# B&R Automation Studio project 8238 (part 11)

```iecst
			//###DK2012Jan12
			// Set statistic.
			IF _wPrevMsgStatisticSelect <> IFmnMsg.In.wMsgStatisticSelect THEN
				_wPrevMsgStatisticSelect := IFmnMsg.In.wMsgStatisticSelect;
				_xMsgStatisticSelectChanged := TRUE;
			END_IF;

			IF IFmnMsg.Trig.xRefreshStatistic OR _xRefreshStatistic THEN
				_msgStatisticNumShowIdx := _msgStatisticNumIdx;
				_msgStatisticTimeShowIdx := _msgStatisticTimeIdx;
				_wIFMsgStatisticCntNumShow := _wIFMsgStatisticCntNum;
				_wIFMsgStatisticCntTimeShow := _wIFMsgStatisticCntTime;
				IFmnMsg.Trig.xRefreshStatistic := FALSE;
				_xRefreshStatistic := FALSE;
				_xMsgStatisticSelectChanged := TRUE;
			END_IF;

			IF _xMsgStatisticSelectChanged THEN
				IF IFmnMsg.In.wMsgStatisticSelect = 0 THEN
					IFmnMsg.Out.wMsgStatisticCnt := _wIFMsgStatisticCntNumShow;
					FOR _wMsgListCnt := 0 TO MNMSG_MAX_IDX_VCMSGSTATLIST BY 1 DO
						_utfMsgTextTempFirst := UINT_TO_WSTRING(_msgStatisticNumShowIdx[_wMsgListCnt].wFunction_ID);
						_utfMsgTextTempSecond := ".";
						brwcsncat(ADR(_utfMsgTextTempFirst), ADR(_utfMsgTextTempSecond),
						UDINT_TO_UINT(brwcslen(ADR(_utfMsgTextTempSecond)) - (brwcslen(ADR(_utfMsgTextTempFirst)) + brwcslen(ADR(_utfMsgTextTempSecond)) - (SIZEOF(_utfMsgTextTempFirst) / 2 - 1))));
						_utfMsgTextTempSecond := UINT_TO_WSTRING(_msgStatisticNumShowIdx[_wMsgListCnt].wMsgNumber);
						brwcsncat(ADR(_utfMsgTextTempFirst), ADR(_utfMsgTextTempSecond),
						UDINT_TO_UINT(brwcslen(ADR(_utfMsgTextTempSecond)) - (brwcslen(ADR(_utfMsgTextTempFirst)) + brwcslen(ADR(_utfMsgTextTempSecond)) - (SIZEOF(_utfMsgTextTempFirst) / 2 - 1))));
						_utfMsgTextTempSecond := ".";
						brwcsncat(ADR(_utfMsgTextTempFirst), ADR(_utfMsgTextTempSecond),
						UDINT_TO_UINT(brwcslen(ADR(_utfMsgTextTempSecond)) - (brwcslen(ADR(_utfMsgTextTempFirst)) + brwcslen(ADR(_utfMsgTextTempSecond)) - (SIZEOF(_utfMsgTextTempFirst) / 2 - 1))));
						_utfMsgTextTempSecond := UINT_TO_WSTRING(_msgStatisticNumShowIdx[_wMsgListCnt].wInstance);
						brwcsncat(ADR(_utfMsgTextTempFirst), ADR(_utfMsgTextTempSecond),
						UDINT_TO_UINT(brwcslen(ADR(_utfMsgTextTempSecond)) - (brwcslen(ADR(_utfMsgTextTempFirst)) + brwcslen(ADR(_utfMsgTextTempSecond)) - (SIZEOF(_utfMsgTextTempFirst) / 2 - 1))));
						_utfMsgTextTempSecond := " ";
						brwcsncat(ADR(_utfMsgTextTempFirst), ADR(_utfMsgTextTempSecond),
						UDINT_TO_UINT(brwcslen(ADR(_utfMsgTextTempSecond)) - (brwcslen(ADR(_utfMsgTextTempFirst)) + brwcslen(ADR(_utfMsgTextTempSecond)) - (SIZEOF(_utfMsgTextTempFirst) / 2 - 1))));
						_wActFunctionID := _msgStatisticNumShowIdx[_wMsgListCnt].wFunction_ID;
						_wActMsgNumber := _msgStatisticNumShowIdx[_wMsgListCnt].wMsgNumber;
						_wActInstance := _msgStatisticNumShowIdx[_wMsgListCnt].wInstance;
						_actGetTxtFim;
						IF NOT((_wActFunctionID = 0) OR (_wActMsgNumber = 0)) THEN
							IFmnMsg.Out.MsgStatistic[_wMsgListCnt].utfMsgText := _utfMsgTextTempFirst;
							IFmnMsg.Out.MsgStatistic[_wMsgListCnt].lValue := _msgStatisticNumShowIdx[_wMsgListCnt].lValue;
						ELSE
							IFmnMsg.Out.MsgStatistic[_wMsgListCnt].utfMsgText := "";
							IFmnMsg.Out.MsgStatistic[_wMsgListCnt].lValue := 0;
						END_IF;
					END_FOR;
				END_IF;
				IF IFmnMsg.In.wMsgStatisticSelect = 1 THEN
					IFmnMsg.Out.wMsgStatisticCnt := _wIFMsgStatisticCntTimeShow;
					FOR _wMsgListCnt := 0 TO MNMSG_MAX_IDX_VCMSGSTATLIST BY 1 DO
						_utfMsgTextTempFirst := UINT_TO_WSTRING(_msgStatisticTimeShowIdx[_wMsgListCnt].wFunction_ID);
						_utfMsgTextTempSecond := ".";
						brwcsncat(ADR(_utfMsgTextTempFirst), ADR(_utfMsgTextTempSecond),
						UDINT_TO_UINT(brwcslen(ADR(_utfMsgTextTempSecond)) - (brwcslen(ADR(_utfMsgTextTempFirst)) + brwcslen(ADR(_utfMsgTextTempSecond)) - (SIZEOF(_utfMsgTextTempFirst) / 2 - 1))));
						_utfMsgTextTempSecond := UINT_TO_WSTRING(_msgStatisticTimeShowIdx[_wMsgListCnt].wMsgNumber);
						brwcsncat(ADR(_utfMsgTextTempFirst), ADR(_utfMsgTextTempSecond),
						UDINT_TO_UINT(brwcslen(ADR(_utfMsgTextTempSecond)) - (brwcslen(ADR(_utfMsgTextTempFirst)) + brwcslen(ADR(_utfMsgTextTempSecond)) - (SIZEOF(_utfMsgTextTempFirst) / 2 - 1))));
						_utfMsgTextTempSecond := ".";
						brwcsncat(ADR(_utfMsgTextTempFirst), ADR(_utfMsgTextTempSecond),
						UDINT_TO_UINT(brwcslen(ADR(_utfMsgTextTempSecond)) - (brwcslen(ADR(_utfMsgTextTempFirst)) + brwcslen(ADR(_utfMsgTextTempSecond)) - (SIZEOF(_utfMsgTextTempFirst) / 2 - 1))));
						_utfMsgTextTempSecond := UINT_TO_WSTRING(_msgStatisticTimeShowIdx[_wMsgListCnt].wInstance);
						brwcsncat(ADR(_utfMsgTextTempFirst), ADR(_utfMsgTextTempSecond),
						UDINT_TO_UINT(brwcslen(ADR(_utfMsgTextTempSecond)) - (brwcslen(ADR(_utfMsgTextTempFirst)) + brwcslen(ADR(_utfMsgTextTempSecond)) - (SIZEOF(_utfMsgTextTempFirst) / 2 - 1))));
						_utfMsgTextTempSecond := " ";
						brwcsncat(ADR(_utfMsgTextTempFirst), ADR(_utfMsgTextTempSecond),
						UDINT_TO_UINT(brwcslen(ADR(_utfMsgTextTempSecond)) - (brwcslen(ADR(_utfMsgTextTempFirst)) + brwcslen(ADR(_utfMsgTextTempSecond)) - (SIZEOF(_utfMsgTextTempFirst) / 2 - 1))));
						_wActFunctionID := _msgStatisticTimeShowIdx[_wMsgListCnt].wFunction_ID;
						_wActMsgNumber := _msgStatisticTimeShowIdx[_wMsgListCnt].wMsgNumber;
						_wActInstance := _msgStatisticTimeShowIdx[_wMsgListCnt].wInstance;
						_actGetTxtFim;
						IF NOT ((_wActFunctionID = 0) OR (_wActMsgNumber = 0)) THEN
							IFmnMsg.Out.MsgStatistic[_wMsgListCnt].utfMsgText := _utfMsgTextTempFirst;
							IFmnMsg.Out.MsgStatistic[_wMsgListCnt].lValue := _msgStatisticTimeShowIdx[_wMsgListCnt].lValue;
						ELSE
							IFmnMsg.Out.MsgStatistic[_wMsgListCnt].utfMsgText := "";
							IFmnMsg.Out.MsgStatistic[_wMsgListCnt].lValue := 0;
						END_IF;
					END_FOR;
				END_IF;
				_xMsgStatisticSelectChanged := FALSE;
			END_IF;
			//###DK2012Jan12

		END_IF

	ELSE	// _Plausibility.xOK

		// Horning for 500ms. After it has finished it will start again ten seconds later.
		_tonCrit1(IN := NOT _tonCrit2.Q, PT := T#500ms);
		_tonCrit2(IN := _tonCrit1.Q, PT := T#10s);

		IFmnMsg.Out.bHorn := SEL(NOT _tonCrit1.Q, 0, 1);	// Causes some horning now.

		IFmnMsg.Out.bLight := 1;

		// Meldung setzen

		IF _xNotOkFirstScan THEN

			_xNotOkFirstScan := FALSE;

			// Meldungsliste füllen

			brsmemset (ADR(mnMsgStatAd.Msg), 0, SIZEOF (mnMsgStatAd.Msg));

			_InsertMsgLine.AdrIntFaultList := ADR(mnMsgStatAd.Msg.MsgListFaultInt);
			_InsertMsgLine.AdrCntIntFault := ADR(mnMsgStatAd.Msg.MsgCntFaultInt);

			_dtHelp(enable := TRUE);

			_InsertMsgLine.Class := MNMSG_CLASS_INTFAULT;
			_InsertMsgLine.Insert := TRUE;
			_InsertMsgLine.MsgLine.bAckLevel := MNMSG_CLASS_NO_ACK;
			_InsertMsgLine.MsgLine.bInstance := 0;
			_InsertMsgLine.MsgLine.diAttr1 := 0;
			_InsertMsgLine.MsgLine.wFunction_ID := 2;
			_InsertMsgLine.MsgLine.wMsgNumber := MNMSG_MSG_SYSTEMFAULT;
			_InsertMsgLine.MsgLine.TimeStamp := _dtHelp.DT1;
			_InsertMsgLine();

			mnMsgStatAd.Msg.dtMsgIntFaultChanged := _dtHelp.DT1;

		END_IF

	END_IF;	// IFmnMsg.Out.xMnMsgReady

	////////////////////////////////////////////////////////////////////////////////////////////////////////////////////////////////////////////////////////////////////////////////////////////////////////////////////////////////////////////////////////////////////////////////////////////////////////////////////////////////////////////////////////////////////////////////////////////////////////////////////////////////////////////////////////////////////////////////////////////////////////////////////////////////////////////////////////////////////////////////////////////////////////////////////////////////////

	_LastExecute(enable := TRUE);
	_dtLastExecute := _LastExecute.DT1;

END_PROGRAM
```

#### mnMsgInit.st - Initialization code
```iecst
(********************************************************************
 * COPYRIGHT -- Herbert Kannegiesser GmbH
 ********************************************************************
 * Program: mnMsg
 * File: mnMsgInit.st
 * Author: subramaniam/hunholz
 * Created: January 28, 2011
 * Changed: October 20, 2011 by A. Hunholz
 ********************************************************************
 * Implementation of program mnMsg
 ********************************************************************
*)
PROGRAM _INIT

	// Packet-Version auslesen mit MO_ver aus SYS_lib und für den Additional Status zur Verfügung stellen

	_sPkgName := 'mnMsg';

	IF ( MO_ver(ADR(_sPkgName), 0, ADR(_VerStruc)) = 0 ) THEN

		brsmemcpy(ADR(mnMsgStatAd.sPkgVersion), ADR(_VerStruc.version), SIZEOF(_VerStruc.version));

	ELSE

		mnMsgStatAd.sPkgVersion := '---';

	END_IF

	//********************Startoption der Plausibilitaetspruefung**********************
	//____________________________________________________________

	// Initialisierung von (Zaehl)variablen und Booleans
	_xMsgStatisticNumFirstEntry 	:= TRUE;
	_xMsgStatisticWriteNum 			:= TRUE;
	_xMsgStatisticTimeFirstEntry 	:= TRUE;
	_xMsgStatisticWriteTime 		:= TRUE;
	_xFirstElementToInsertTime 		:= TRUE;
	_xFirstElementToInsertNum 		:= TRUE;

	// Filter setzen
	IFmnMsg.In.wMsgHistListClassSelect.0 := 1;
	IFmnMsg.In.wMsgHistListClassSelect.1 := 1;
	IFmnMsg.In.wMsgHistListClassSelect.2 := 1;
	IFmnMsg.In.wMsgHistListClassSelect.3 := 1;

	_EventStatisticDelStep := Del_Wait;

	//*********************Synchrone Schnittstelle zurücksetzen*****************************

	brsmemset(ADR(IFmnMsg.Out),0,SIZEOF(IFmnMsg.Out));
	brsmemset (ADR (kgMsgStatus[MNMSG_IDX_KGMSGSTAT]), 0, SIZEOF (kgMsgStatus[0]));

	//*********************Alle Listen loeschen

	brsmemset (ADR(_MsgImage), 0, SIZEOF (_MsgImage));	// Meldungsabbild
	brsmemset (ADR(_MsgImageState),0,SIZEOF(_MsgImageState));	// Meldungsabbild

	brsmemset (ADR(mnMsgStatAd.Msg), 0 ,SIZEOF (mnMsgStatAd.Msg));

	//****************************************************************************************************************
	// Log erzeugen
	//****************************************************************************************************************

	_kgArLogWrite.enable := TRUE;
	_kgArLogWrite.ident := 0;
	_kgArLogWrite.errornr := 50001;

	_AsArLogCreate(enable := TRUE, pName := ADR('mnMsgL'), len := 4096, memType := arlogUSRROM);

	IF _AsArLogCreate.status = ERR_OK THEN

		_kgArLogWrite.ident := _AsArLogCreate.ident;

	ELSIF _AsArLogCreate.status = arlogERR_EXISTING THEN

		_AsArLogGetInfo(enable := TRUE, pName := ADR('mnMsgL'));

		IF _AsArLogGetInfo.status = ERR_OK THEN

			_kgArLogWrite.ident := _AsArLogGetInfo.ident;

		END_IF

	END_IF

	//***************** Datenobjekte prüfen
	//______________________________

	// Unbedingtes REPEAT, damit bei Fehler alles Andere per EXIT
	// übersprungen werden kann.

	REPEAT

		//*************** KONFIGURATION
		//**************************************
		// _doInfoCfg 'Bild der Konfigurationsdatei' of DatObjInfo

		_doInfoCfg.enable := TRUE;	// VAR_INPUT BOOL enable 'enables execution'
		_doInfoCfg.pName := ADR('CfgMsgStat');	// VAR_INPUT UDINT pName 'name of data object'
		_doInfoCfg();

		IF _doInfoCfg.status <> ERR_OK THEN

			_kgArLogWrite.logLevel := arlogLEVEL_INFO;
			_kgArLogWrite.text := 'Messageconfiguration does not exist: {##AttrVar1}';
			_kgArLogWrite.var1 := _doInfoCfg.status;
			_kgArLogWrite.var2 := 0;
			_kgArLogWrite();
			EXIT;

		ELSE

			// _doInfoCfg 'Bild der Konfigurationsdatei' of DatObjInfo
			// wCntCfg of Plausib_Typ: number of configuration entries
			_Plausibility.dCfgLen := _doInfoCfg.len; // VAR_OUTPUT UDINT len 'length of the data area in the data object'
			_Plausibility.dCfgMem := _doInfoCfg.pDatObjMem; // VAR_OUTPUT UDINT pDatObjMem 'pointer to the data in the data object'
			_Plausibility.wCfgCnt := UDINT_TO_UINT((_doInfoCfg.len-SIZEOF(UINT))/SIZEOF (MsgCfgLine_Typ)); // Laenge der Version zu Beginn abziehen

			_wVersion ACCESS _Plausibility.dCfgMem;
			_Plausibility.wCfgVersion := _wVersion;

			IF _Plausibility.wCfgCnt > MNMSG_MAX_CFGMESSAGES THEN

				_kgArLogWrite.logLevel := arlogLEVEL_INFO;
				_kgArLogWrite.text := 'To much entries in Messageconfiguration: {##AttrVar1}';
				_kgArLogWrite.var1 := _Plausibility.wCfgCnt;
				_kgArLogWrite.var2 := 0;
				_kgArLogWrite();
				EXIT;

			END_IF

			// Zugriff auf die Konfigurationszeilen
			_MsgCfgList ACCESS _doInfoCfg.pDatObjMem + SIZEOF(UINT); // Offset Versionsnummer

			// Binäre Suche initialisieren
			_BinSearchCfg.MsgCfgList := _doInfoCfg.pDatObjMem + SIZEOF(UINT);	// Offset Versionsnummer
			_BinSearchCfg.wCntMsgCfg := _Plausibility.wCfgCnt;	// VAR_INPUT UINT wCntMsgCfg

		END_IF

		//*****************************
		// STATISTIK
		//*****************************

		_kgCheckStat(Enable := TRUE, pName := ADR('_MsgStat'), MinLen := SIZEOF(_MsgStatList), NomLen := SIZEOF(_MsgStatList), Create := TRUE, MemType := doUSRROM);

		IF _kgCheckStat.Status = ERR_OK OR _kgCheckStat.Status = KG_INFO_DO_NEW THEN

			_doWriteStat.enable := TRUE;
			_doWriteStat.ident := _kgCheckStat.doId;

			IF _kgCheckStat.Status = KG_INFO_DO_NEW THEN

				// Kopfdaten schreiben
				_StatHeader.lVersion := _Plausibility.wCfgVersion;
				_StatHeader.lLength :=  UINT_TO_UDINT(MNMSG_MAX_CFGMESSAGES);

				_doWriteStat.Offset := 0;
				_doWriteStat.len := SIZEOF(_StatHeader);
				_doWriteStat.pSource := ADR(_StatHeader);
				_doWriteStat();

				IF _doWriteStat.status = ERR_OK THEN

					_xStatReady := TRUE;
					_MsgStatList ACCESS _kgCheckStat.doMem;

					_kgArLogWrite.logLevel := arlogLEVEL_INFO;
					_kgArLogWrite.text := 'Statistic created!';
					_kgArLogWrite.var1 := 0;
					_kgArLogWrite.var2 := 0;
					_kgArLogWrite();

				ELSE

					_kgArLogWrite.logLevel := arlogLEVEL_INFO;
					_kgArLogWrite.text := 'Write Statistic: {##AttrVar1}';
					_kgArLogWrite.var1 := _doWriteStat.status;
					_kgArLogWrite.var2 := 0;
					_kgArLogWrite();

				END_IF

			ELSE

				brsmemcpy(ADR(_StatHeader), _kgCheckStat.doMem, SIZEOF(_StatHeader));

				IF _StatHeader.lVersion <> _Plausibility.wCfgVersion THEN

					//Konfigurationsversion hat sich geändert --> Statistik neu erstellen

					_doDeleteStat(enable := TRUE, ident := _kgCheckStat.doId);

					_kgCheckStat(Enable := TRUE, pName := ADR('_MsgStat'), MinLen := SIZEOF(_MsgStatList), NomLen := SIZEOF(_MsgStatList), Create := TRUE, MemType := doUSRROM);

					IF _kgCheckStat.Status = KG_INFO_DO_NEW THEN

						_doWriteStat.enable := TRUE;
						_doWriteStat.ident := _kgCheckStat.doId;

						// Kopfdaten schreiben
						_StatHeader.lVersion := _Plausibility.wCfgVersion;
						_StatHeader.lLength :=  UINT_TO_UDINT(MNMSG_MAX_CFGMESSAGES);

						_doWriteStat.Offset := 0;
						_doWriteStat.len := SIZEOF(_StatHeader);
						_doWriteStat.pSource := ADR(_StatHeader);
						_doWriteStat();

						IF _doWriteStat.status = ERR_OK THEN

							_xStatReady := TRUE;
							_MsgStatList ACCESS _kgCheckStat.doMem;

							_kgArLogWrite.logLevel := arlogLEVEL_INFO;
							_kgArLogWrite.text := 'Statistic recreated!';
							_kgArLogWrite.var1 := 0;
							_kgArLogWrite.var2 := 0;
							_kgArLogWrite();

						ELSE

							_kgArLogWrite.logLevel := arlogLEVEL_INFO;
							_kgArLogWrite.text := 'Write Statistic*: {##AttrVar1}';
							_kgArLogWrite.var1 := _doWriteStat.status;
							_kgArLogWrite.var2 := 0;
							_kgArLogWrite();

						END_IF

					ELSE

						_kgArLogWrite.logLevel := arlogLEVEL_INFO;
						_kgArLogWrite.text := 'Check Statistic*: {##AttrVar1}';
						_kgArLogWrite.var1 := _kgCheckStat.Status;
						_kgArLogWrite.var2 := 0;
						_kgArLogWrite();

					END_IF

				ELSE //IF _StatHeader.lVersion <> _Plausibility.wCfgVersion THEN

					// Version ist OK
					_xStatReady := TRUE;
					_MsgStatList ACCESS _kgCheckStat.doMem;

				END_IF

			END_IF

		ELSE

			_kgArLogWrite.logLevel := arlogLEVEL_INFO;
			_kgArLogWrite.text := 'Check Statistic: {##AttrVar1}';
			_kgArLogWrite.var1 := _kgCheckStat.Status;
			_kgArLogWrite.var2 := 0;
			_kgArLogWrite();

		END_IF

		//*************** RINGBUFFER
		//*********************************

		_kgCheckHist(Enable := TRUE, pName := ADR('_MsgRB'), MinLen :=  MNMSG_MAX_MESSAGEHISTORY * SIZEOF(MsgHistList_Typ), NomLen :=  MNMSG_MAX_MESSAGEHISTORY * SIZEOF(MsgHistList_Typ), Create := TRUE, MemType := doUSRROM);

		IF _kgCheckHist.Status = ERR_OK OR _kgCheckHist.Status = KG_INFO_DO_NEW THEN

			IF _kgCheckHist.Status = KG_INFO_DO_NEW THEN

				_kgArLogWrite.logLevel := arlogLEVEL_INFO;
				_kgArLogWrite.text := 'History created!';
				_kgArLogWrite.var1 := 0;
				_kgArLogWrite.var2 := 0;
				_kgArLogWrite();

				_wPtrRBwrite := 0;
				_wPtrRBread := 0;
				_wPtrRBloc := 0;

			END_IF

			_xRBReady := TRUE;

			// _InsertRB of msgInsertRB 'Eintrag in den Ringbuffer'
			_InsertRB.doIdent := _kgCheckHist.doId;
			_InsertRB.doLen := _kgCheckHist.doLen;

			_ReadRB.doIdent := _kgCheckHist.doId;
			_ReadRB.doLen := _kgCheckHist.doLen;

			_LocRB.doIdent := _kgCheckHist.doId;
			_LocRB.doLen := _kgCheckHist.doLen;

			_DebugHistory ACCESS _kgCheckHist.doMem;

		ELSE

			_kgArLogWrite.logLevel := arlogLEVEL_INFO;
			_kgArLogWrite.text := 'Check History: {##AttrVar1}';
			_kgArLogWrite.var1 := _kgCheckStat.Status;
			_kgArLogWrite.var2 := 0;
			_kgArLogWrite();

		END_IF

		_Plausibility.xOK := TRUE;

		//***********************************************************************************
		// Statistik für Werte vor dem letzten Ausschalten schreiben, um dann die
		// Statistik zurücksetzen zu können
		//***********************************************************************************

		IF _xRBReady THEN

			FOR _wMsgIdx := 1 TO _Plausibility.wCfgCnt DO

				IF _MsgImageTime[_wMsgIdx].dtTimeStamp <> DT#1970-01-01-00:00:00  THEN

					// Es steht noch eine Zeit im Image, die noch nicht erfasst wurde
					// D.h. beim Ausschalten der SPS stand diese Meldung noch an.

					_lTime := 0;

					IF _xStatReady THEN

						// Statistik schreiben
						IF (_dtLastExecute >= _MsgImageTime[_wMsgIdx].dtTimeStamp) THEN
							_lTime := DiffDT(_dtLastExecute, _MsgImageTime[_wMsgIdx].dtTimeStamp);
						END_IF

						_StatLine.lTime := _MsgStatList.List[_wMsgIdx].lTime + _lTime;
						_StatLine.lCnt := _MsgStatList.List[_wMsgIdx].lCnt + 1;
						_StatLine.wFunction_ID := _MsgCfgList[_wMsgIdx].wFunction_ID;
						_StatLine.wMsgNumber := _MsgCfgList[_wMsgIdx].wMsgNumber;
						_StatLine.wInstance := _MsgCfgList[_wMsgIdx].wInstance;
						_StatLine.wMsgClass := _MsgStatList.List[_wMsgIdx].wMsgClass;

						_doWriteStat.Offset := SIZEOF(_StatHeader) + (_wMsgIdx-1)*SIZEOF(_StatLine);
						_doWriteStat.len := SIZEOF(_StatLine);
						_doWriteStat.pSource := ADR(_StatLine);

						_doWriteStat();

					END_IF

					// Ringbuffer schreiben
					_TempHistline.TimeStampEvent := _dtLastExecute;
					_TempHistline.wFunction_ID := _MsgCfgList[_wMsgIdx].wFunction_ID;
					_TempHistline.wInstance := _MsgCfgList[_wMsgIdx].wInstance;
					_TempHistline.wMsgNumber := _MsgCfgList[_wMsgIdx].wMsgNumber;
					IF _xStatReady THEN
						_TempHistline.wMsgClass := _MsgStatList.List[_wMsgIdx].wMsgClass;
					ELSE
						_TempHistline.wMsgClass := MNMSG_CLASS_INFO;
					END_IF
					_TempHistline.diAttr1 := 0;
					_TempHistline.diAttr2 := 0;
					_TempHistline.sAttrTxt := '';
					_TempHistline.wEvent := MNMSG_EVENT_GONE;	// Constant of library KGlibMMsg UINT MSG_EVENT_GONE = 3
					_TempHistline.lTime := _lTime;

					_InsertRB.pEntry := ADR(_TempHistline);
					_InsertRB.lLenEntry := SIZEOF(_TempHistline);
					_InsertRB(wPtrWrite := _wPtrRBwrite, wPtrRead := _wPtrRBread, wPtrStart := _wPtrRBstart);

					IF _InsertRB.wStatus <> ERR_OK THEN
						_kgArLogWrite.logLevel := arlogLEVEL_INFO;
						_kgArLogWrite.text := 'Inster History: {##AttrVar1}';
						_kgArLogWrite.var1 := _InsertRB.wStatus;
						_kgArLogWrite.var2 := 0;
						_kgArLogWrite();
					END_IF

				END_IF

			END_FOR

		END_IF

		// Nachdem das Image in die Statistik und in den Ringbuffer geschrieben wurde,
		// kann es auf Null zurückgesetzt werden
		brsmemset(ADR(_MsgImageTime),0,SIZEOF(_MsgImageTime));

		UNTIL

		TRUE

	END_REPEAT;

	_dtHelp(enable := TRUE);

	_xStatFault := NOT _xStatReady;

	_xNotOkFirstScan := TRUE;

END_PROGRAM
```

#### mnMsg.typ - Local data types
```iecst
(********************************************************************
 * COPYRIGHT -- Herbert Kannegiesser GmbH
 ********************************************************************
 * Program: mnMsg
 * File: mnMsg.typ
 * Author: subramaniam/Hunholz
 * Created: January 28, 2011
 * Changed: June 15, 2011
 ********************************************************************
 * Local data types of program mnMsg
 ********************************************************************)

TYPE
	CmdState_enum :
		(
		enCS_Idle,
		enCS_WaitForZero,
		enCS_CmdDelStat,
		enCS_CmdDelHist
		);
	EventStatisticDel_enum :
		(
		Del_Delete,
		Del_Wait,
		Del_Check,
		Del_Write,
		Del_Error
		);
	EventHistDel_enum :
		(
		Del_DeleteH,
		Del_WaitH,
		Del_ErrorH
		);
END_TYPE

(*Plausibilitaetspruefung Meldungsmanager ----------------------------------------------------------------------------------------------------------------------------------------------------------------------------------------*)

TYPE
	Plausib_Typ : 	STRUCT
		dCfgMem : UDINT;
		dCfgLen : UDINT;
		wCfgCnt : UINT;
		wCfgVersion : UINT;
		xOK : BOOL;
	END_STRUCT;
END_TYPE

(*Meldungsabbild ----------------------------------------------------------------------------------------------------------------------------------------------------------------------------------------*)

TYPE
	ImageMsgState_Typ : 	STRUCT
		xOn : BOOL;
		xChanged : BOOL;
	END_STRUCT;
	ImageMsgTime_Typ : 	STRUCT
		dtTimeStamp : DATE_AND_TIME;
	END_STRUCT;
	ImageMsg_Typ : 	STRUCT
		wStatus : UINT;
		wMsgClass : UINT;
		wMsgAckLevel : UINT;
		sMsgAttrTxt : STRING[13];
		diMsgAttr1 : DINT;
		diMsgAttr2 : DINT;
	END_STRUCT;
	ImageMsgHelp_Typ : 	STRUCT  (*Hilfsstruktur der Meldeabbild*)
		xFaultIntChanged : BOOL;
		xFaultExtChanged : BOOL;
		xWarningChanged : BOOL;
		xInfoChanged : BOOL;
		xMaintChanged : BOOL;
	END_STRUCT;
	mnMsgStatisticIdx_Type : 	STRUCT
		wFunction_ID : UINT;
		wMsgNumber : UINT;
		wInstance : UINT;
		lValue : UDINT;
	END_STRUCT;
END_TYPE
```

#### mnMsg.var - Local variables
```iecst
(********************************************************************
 * COPYRIGHT -- Herbert Kannegiesser GmbH
 ********************************************************************
 * Program: mnMsg
 * File: mnMsg.var
 * Author: subramaniam/hunholz
 * Created: January 28, 2011
 * Changed: June 15, 2011
 ********************************************************************
 * Local variables of program mnMsg
 ********************************************************************)
(*Plausibilitaetspruefung Meldungsmanager *)
VAR
	_Plausibility : Plausib_Typ := (dCfgMem:=0,dCfgLen:=0,wCfgCnt:=0,wCfgVersion:=0,xOK:=FALSE);
	_xTrigRefreshHistList : BOOL;
	_lErrCnt : UDINT;
	_TONrepeatDFII : TON;
END_VAR
(*Meldungsabbild *)
VAR
	_MsgImage : ARRAY[1..MNMSG_MAX_CFGMESSAGES] OF ImageMsg_Typ;
	_MsgImageState : ARRAY[1..MNMSG_MAX_CFGMESSAGES] OF ImageMsgState_Typ;
	_MsgImageHelp : ImageMsgHelp_Typ;
END_VAR
VAR RETAIN
	_MsgImageTime : ARRAY[1..MNMSG_MAX_CFGMESSAGES] OF ImageMsgTime_Typ;
END_VAR
(* Bild der Konfigurationsdatei *)
VAR
	_doInfoCfg : DatObjInfo;
	_MsgCfgList : REFERENCE TO ARRAY[1..MNMSG_MAX_CFGMESSAGES] OF MsgCfgLine_Typ;
END_VAR
(*Bild der Textdatei*)
(* In diesem Fall, wird die Länge des Arrays nicht von mnTxt bestimmt *)
VAR
	_MsgTxtLine : REFERENCE TO ARRAY[1..MNMSG_MAX_CFGMESSAGES] OF MsgTxtLine_Typ;
	_MsgHelpTxtLine : REFERENCE TO ARRAY[1..MNMSG_MAX_CFGMESSAGES] OF MsgHelpTxtLine_Typ;
END_VAR
(* Bild der Statistikdatei*)
VAR
	_MsgStatList : REFERENCE TO MsgStat_Typ;
END_VAR
(*Bild der Text-Meldungshistorie*)
VAR
	_MsgHistListRB : ARRAY[0..MNMSG_MAX_IDX_VCMSGHISTLIST] OF IFmnMsgOutMsgHistList_Typ;
END_VAR
(*Interne Meldung*)
VAR
	_mnMsgStat : kgMsg_Status_Typ := (0);
END_VAR
(*Kommandbefehle *)
(*  Zeiger auf Zusatzattribute *)
VAR
	_iCmdData0 : REFERENCE TO ARRAY[0..1] OF UINT;
	_iCmdData1 : REFERENCE TO ARRAY[0..1] OF UINT;
END_VAR
(*Schnittstelle Visualisierung für Ringbuffer und Statistik *)
VAR
	_xAck : BOOL;
	_wCntFaultNotAck : UINT;
	_xCmdAckAll : BOOL;
	_xCmdAck : BOOL;
	_xCmdAckAllMaint : BOOL;
END_VAR
(*Letzte Ausführungszeit bestimmen*)
VAR
	_LastExecute : DTGetTime;
END_VAR
VAR RETAIN
	_dtLastExecute : DATE_AND_TIME := 0;
END_VAR
(*Aktueller Zeitstempel*)
VAR
	_dtTimeStamp : DTGetTime;
END_VAR
(* Binäre Suche *)
VAR
	_BinSearchCfg : msgBinSearchCfgList;
	_BinSearchTxt : msgBinSearchTxtLine;
	_BinSearchHelpTxt : msgBinSearchHelpTxtLine;
END_VAR
(*Suche*)
VAR
	_GetNextChrPos : msgNextChrPos;
END_VAR
(* Ringbuffer *)
VAR
	_InsertRB : kgRBinsert;
	_ReadRB : kgRBread;
	_LocRB : kgRBloc;
	_wStepRdRb : UINT;
	_xRBReady : BOOL := FALSE;
	_xMnTxtReady : BOOL := FALSE;
END_VAR
VAR RETAIN
	_wPtrRBwrite : UINT;
	_wPtrRBread : UINT;
	_wPtrRBloc : UINT;
	_wPtrRBstart : UINT;
END_VAR
(* Statistik*)
VAR
	_StatLine : MsgStatList_Typ;
	_StatHeader : MsgStatHeader_Typ;
	_doWriteStat : DatObjWrite;
	_doDeleteStat : DatObjDelete;
	_xStatReady : BOOL := FALSE;
END_VAR
(* Meldungslisten *)
VAR
	_InsertMsgLine : msgInsertMsgLine;
END_VAR
(* Hupensteuerung *)
VAR
	_xHornFaultOn : BOOL;
	_xHornWarnOn : BOOL;
	_tpFault : TP;
	_tonFault1 : TON;
	_tonFault2 : TON;
	_xHornFaultOnh : BOOL;
	_xHornWarnOnh : BOOL;
	_tpWarn : TP;
	_tonWarn2 : TON;
	_tonWarn1 : TON;
	_wFaultMode : UINT;
	_wWarnMode : UINT;
END_VAR
(*MsgStatistic*)
VAR
	_msgStatisticNumIdx : ARRAY[0..MNMSG_MAX_IDX_VCMSGSTATLIST] OF mnMsgStatisticIdx_Type;
	_msgStatisticTimeIdx : ARRAY[0..MNMSG_MAX_IDX_VCMSGSTATLIST] OF mnMsgStatisticIdx_Type;
	_msgStatisticNumShowIdx : ARRAY[0..MNMSG_MAX_IDX_VCMSGSTATLIST] OF mnMsgStatisticIdx_Type;
	_msgStatisticTimeShowIdx : ARRAY[0..MNMSG_MAX_IDX_VCMSGSTATLIST] OF mnMsgStatisticIdx_Type;
END_VAR
(* Hilfsvariablen *)
VAR
	_wSrcIdx : UDINT;
	_wMsgIdx : UINT;
	_wTxtIdx : UINT;
	_wImageIdx : UINT;
	_lTime : UDINT;
	_ii : UINT;
	_dtHelp : DTGetTime;
	_xMnParOk : BOOL := FALSE;
	_xMsgClassChanged : BOOL := FALSE;
	_xAckLevelChanged : BOOL;
	_xAckLevelRosen : BOOL := FALSE;
	_xAckLevelFallen : BOOL := FALSE;
	_EventStatisticDelStep : EventStatisticDel_enum;
	_EventHistDelStep : EventHistDel_enum;
	_tonCrit1 : TON;
	_tonCrit2 : TON;
END_VAR
VAR CONSTANT
	MSW : UINT := 1; (*Most Significant Word*)
	LSW : UINT := 0; (*Leas Significant Word*)
END_VAR
VAR
	_enIFCmdState : CmdState_enum := enCS_Idle;
	_enExtCmdState : CmdState_enum := enCS_Idle;
	_xIFcmdHornOff : BOOL := FALSE;
	_wMsgListCnt : UINT;
	_wIFMsgListCnt : UINT;
	_wIFMsgStatisticCntTime : UINT;
	_wIFMsgStatisticCntNum : UINT;
	_wIFMsgStatisticCntTimeShow : UINT;
	_wIFMsgStatisticCntNumShow : UINT;
	_xMsgStatisticNumFirstEntry : BOOL;
	_xMsgStatisticWriteNum : BOOL;
	_xMsgStatisticTimeFirstEntry : BOOL;
	_xMsgStatisticWriteTime : BOOL;
	_wPosMinTime : UINT;
	_wPosMinNum : UINT;
	_wPosMaxTime : UINT;
	_wPosMaxNum : UINT;
	_wPosEndTime : UINT;
	_wPosEndNum : UINT;
	_wPosSearchTime : UINT;
	_wPosSearchNum : UINT;
	_diMemMoveTimeIdx : DINT := 0;
	_diMemMoveNumIdx : DINT := 0;
	_xPosFoundTime : BOOL;
	_xPosFoundNum : BOOL;
	_xFirstElementToInsertTime : BOOL;
	_xFirstElementToInsertNum : BOOL;
	_lValueNumMin : UDINT;
	_lValueTimeMin : UDINT;
	_lValueTime : UDINT;
	_lValueNum : UDINT;
	_wPrevMsgStatisticSelect : UINT := 0;
	_xMsgStatisticSelectChanged : BOOL := FALSE;
	_utfMsgTextTempFirst : WSTRING[67];
	_utfMsgTextTempSecond : WSTRING[255];
	_utfMsgTextTempThird : WSTRING[255];
	_utfMsgTextTempFourth : WSTRING[255];
	_fbMsgReplSubStr : msgReplSubStr;
	_lHElseTime1 : UDINT := 0;
	_lHElseTime2 : UDINT := 0;
	_lHElseTime3 : UDINT := 0;
	_lHElseTime3EndPos : UDINT := 0;
	_wHElseTime3PosSearch : UINT := 0;
	_lHElseTime3lValuePosP0 : UDINT := 0;
	_lHElseTime3lValuePosP1 : UDINT := 0;
	_lHElseTime3lValueTime : UDINT := 0;
	_lHElseNum1 : UDINT := 0;
	_lHElseNum2 : UDINT := 0;
	_lHElseNum3 : UDINT := 0;
	_TempHistline : MsgHistList_Typ;
	_kgArLogWrite : kgArLogWrite;
	_AsArLogCreate : AsArLogCreate;
	_AsArLogGetInfo : AsArLogGetInfo;
	_xLogNoCfg : BOOL;
	_xLogCfgMoved : BOOL;
END_VAR
VAR CONSTANT
	MNMSG_MSG_NO_MESSAGE : UINT := 0;
END_VAR
VAR
	_xStatFault : BOOL;
	_xLogDeleteStat : BOOL;
	_xLogCreateStat : BOOL;
	_xLogInfoStat : BOOL;
	_xLogWriteStat : BOOL;
	_wPrevLCID : UINT := 0;
	_xUpdateMsgList : BOOL := FALSE;
	_xUpdateMsgHistListRB : BOOL := FALSE;
	_wMsgHistListCntUpdate : UINT := 0;
	_utfMsgTxtLCIDfirst : WSTRING[67];
	_utfMsgTxtLCIDsecond : WSTRING[67];
	_utfRbsDateTime : WSTRING[67];
	_utfLCIDFunctionId : WSTRING[67];
	_utfLCIDMsgNumber : WSTRING[67];
	_utfLCIDInstance : WSTRING[67];
	_wLCIDFunctionId : UINT;
	_wLCIDMsgNumber : UINT;
	_wLCIDInstance : UINT;
	_lPosPointFirst : UDINT;
	_lPosPointSecond : UDINT;
	_lPosSpaceFirst : UDINT;
	_lPosSpaceSecond : UDINT;
	_lAdrPointFirst : UDINT;
	_lAdrPointSecond : UDINT;
	_lAdrSpaceFirst : UDINT;
	_lAdrSpaceSecond : UDINT;
	_wCntSafety : UINT := 0;
	_sPkgName : STRING[10];
	_VerStruc : MoVerStruc_typ;
	_wPrevMsgHistListOffsetRB : UINT;
	_wMsgHistListOffsetRB : UINT;
	_xRefreshHistListRB : BOOL;
	_xMsgHistListOffsetChRB : BOOL;
	_wPrevMsgHistListEventSelRB : UINT;
	_wMsgHistListEventSelRB : UINT;
	_xMsgHistListEventSelChRB : BOOL;
	_wPrevMsgHistListClassSelRB : UINT;
	_wMsgHistListClassSelRB : UINT;
	_xMsgHistListClassSelChRB : BOOL;
	_xMsgHistListPointToMinRB : BOOL;
	_wPtrRBlocTemp : UINT;
	_wPtrRBlocTempTwo : UINT;
	_wPtrRBlocTempThree : UINT;
	_wPtrRBlocTempFour : UINT;
	_xPtrRBlocAgain : BOOL;
	_wPtrRBlocLastFound : UINT;
	_wMsgHistListMaxOffsetRB : UINT;
	_xTrigPrevMsgHistListPageRB : BOOL;
	_xTrigNextMsgHistListPageRB : BOOL;
	_xRBoneTurn : BOOL;
	_wMsgHistListCntRB : UINT;
	_wActFunctionID : UINT;
	_wActMsgNumber : UINT;
	_diActAttr1 : DINT;
	_diActAttr2 : DINT;
	_sActAttrTxt : STRING[13];
	_wActInstance : UINT;
	_wActEvent : UINT;
	_lActTime : UDINT;
	_bActMsgLClass : USINT;
	_xSelOk : BOOL;
	_xTurnaround : BOOL;
	_xExtCmdAckAll : BOOL;
	_xExtCmdAck : BOOL;
	_xExtCmdAckAllMaint : BOOL;
	_wExtCmdFunctionID : UINT;
	_wExtCmdMsgNo : UINT;
	_wExtCmdInstance : UINT;
	_wExtCmdAckLevel : UINT;
	_xExtcmdHornOff : BOOL;
	_xDeleteMsgStat : BOOL;
	_wMsgCntMaint : UINT;
	_wIdxMsgListMaint : UINT;
	_xUpdateMsgListLan : BOOL;
	_xRefreshStatistic : BOOL;
	_xRefreshHistList : BOOL;
	_wLCID : UINT;
	_kgCheckStat : kgCheckDo;
	_kgCheckHist : kgCheckDo;
	_wVersion : REFERENCE TO UINT;
	_wLogStep : UINT;
	_xNotOkFirstScan : BOOL;
	_DebugHistory : REFERENCE TO ARRAY[0..MNMSG_MAX_MESSAGEHISTORY] OF MsgHistList_Typ;
END_VAR
```

#### _actGetTxtFim.st
```iecst
(********************************************************************
 * COPYRIGHT -- Herbert Kannegiesser GmbH
 ********************************************************************
 * Program: mnMsg
 * File: actGetTxtFim.st
 * Author: kuehne
 * Created: February 21, 2012
 ********************************************************************
 * Implementation of program mnMsg
 ********************************************************************)

(* Add a new action to your IEC program or library *)
ACTION _actGetTxtFim:
	IF _xMnTxtReady THEN
		_MsgTxtLine ACCESS IFmnTxt.Out.ptrFunctionTxtList;
		_BinSearchTxt.MsgTxtList := IFmnTxt.Out.ptrFunctionTxtList;
		_BinSearchTxt.wCntMsgTxt := IFmnTxt.Out.wCntFunctionTxt;
		_BinSearchTxt.wFunctionID := _wActFunctionID;
		_BinSearchTxt.wNumber := _wActMsgNumber;
		_BinSearchTxt.wInstance := _wActInstance;
		_BinSearchTxt.bTupel := 1;
		_BinSearchTxt();
		IF _BinSearchTxt.wStatus <> ERR_OK THEN
			brwcscat(ADR(_utfMsgTextTempFirst), ADR(""));
		ELSE
			_wTxtIdx := _BinSearchTxt.wMsgPos;
			_BinSearchCfg.wFunctionID := _wActFunctionID;
			_BinSearchCfg.wMsgNo := _wActMsgNumber;
			_BinSearchCfg.wInstance := _wActInstance;
			_BinSearchCfg();
			IF _BinSearchCfg.wStatus = ERR_OK THEN
				_wImageIdx := _BinSearchCfg.wMsgIdx;
				_utfMsgTextTempThird := "";
				_utfMsgTextTempThird := DINT_TO_WSTRING(_MsgImage[_wImageIdx].diMsgAttr1);
			ELSE
				_utfMsgTextTempThird := "{##AttrVar1}";
			END_IF;
			_utfMsgTextTempSecond := "";
			_fbMsgReplSubStr.utfStr := ADR(_MsgTxtLine[_wTxtIdx].utfText);
			_fbMsgReplSubStr.utfSubStr := ADR("{##AttrVar1}");
			_fbMsgReplSubStr.utfStrToReplWith := ADR(_utfMsgTextTempThird);
			_fbMsgReplSubStr.utfStrResult := ADR(_utfMsgTextTempSecond);
			_fbMsgReplSubStr();
			IF _BinSearchCfg.wStatus = ERR_OK THEN
				_wImageIdx := _BinSearchCfg.wMsgIdx;
				_utfMsgTextTempThird := "";
				_utfMsgTextTempThird := DINT_TO_WSTRING(_MsgImage[_wImageIdx].diMsgAttr2);
			ELSE
				_utfMsgTextTempThird := "{##AttrVar2}";
			END_IF;
			_utfMsgTextTempFourth := "";
			_utfMsgTextTempFourth := _utfMsgTextTempSecond;
			_utfMsgTextTempSecond := "";
			_fbMsgReplSubStr.utfStr := ADR(_utfMsgTextTempFourth);
			_fbMsgReplSubStr.utfSubStr := ADR("{##AttrVar2}");
			_fbMsgReplSubStr.utfStrToReplWith := ADR(_utfMsgTextTempThird);
			_fbMsgReplSubStr.utfStrResult := ADR(_utfMsgTextTempSecond);
			_fbMsgReplSubStr();
			IF _BinSearchCfg.wStatus = ERR_OK THEN
				_wImageIdx := _BinSearchCfg.wMsgIdx;
				_utfMsgTextTempThird := "";
				_utfMsgTextTempThird := STRING_TO_WSTRING(_MsgImage[_wImageIdx].sMsgAttrTxt);
			ELSE
				_utfMsgTextTempThird := "{##AttrTxt}";
			END_IF;
			_utfMsgTextTempFourth := "";
			_utfMsgTextTempFourth := _utfMsgTextTempSecond;
			_utfMsgTextTempSecond := "";
			_fbMsgReplSubStr.utfStr := ADR(_utfMsgTextTempFourth);
			_fbMsgReplSubStr.utfSubStr := ADR("{##AttrTxt}");
			_fbMsgReplSubStr.utfStrToReplWith := ADR(_utfMsgTextTempThird);
			_fbMsgReplSubStr.utfStrResult := ADR(_utfMsgTextTempSecond);
			_fbMsgReplSubStr();
			brwcsncat(ADR(_utfMsgTextTempFirst), ADR(_utfMsgTextTempSecond),
			UDINT_TO_UINT(brwcslen(ADR(_utfMsgTextTempSecond)) - (brwcslen(ADR(_utfMsgTextTempFirst)) + brwcslen(ADR(_utfMsgTextTempSecond)) - (SIZEOF(_utfMsgTextTempFirst) / 2 - 1))));
			_utfMsgTextTempSecond := "";
			_utfMsgTextTempSecond := ": ";
			brwcsncat(ADR(_utfMsgTextTempFirst), ADR(_utfMsgTextTempSecond),
			UDINT_TO_UINT(brwcslen(ADR(_utfMsgTextTempSecond)) - (brwcslen(ADR(_utfMsgTextTempFirst)) + brwcslen(ADR(_utfMsgTextTempSecond)) - (SIZEOF(_utfMsgTextTempFirst) / 2 - 1))));
		END_IF;
		_MsgTxtLine ACCESS IFmnTxt.Out.ptrInstanceTxtList;
		_BinSearchTxt.MsgTxtList := IFmnTxt.Out.ptrInstanceTxtList;
		_BinSearchTxt.wCntMsgTxt := IFmnTxt.Out.wCntInstanceTxt;
		_BinSearchTxt.wFunctionID := _wActFunctionID;
		_BinSearchTxt.wNumber := _wActInstance;
		_BinSearchTxt.wInstance := 0;
		_BinSearchTxt.bTupel := 2;
		_BinSearchTxt();
		IF _BinSearchTxt.wStatus <> ERR_OK THEN
			brwcscat(ADR(_utfMsgTextTempFirst), ADR(""));
		ELSE
			_wTxtIdx := _BinSearchTxt.wMsgPos;
			_BinSearchCfg.wFunctionID := _wActFunctionID;
			_BinSearchCfg.wMsgNo := _wActMsgNumber;
			_BinSearchCfg.wInstance := _wActInstance;
			_BinSearchCfg();
			IF _BinSearchCfg.wStatus = ERR_OK THEN
				_wImageIdx := _BinSearchCfg.wMsgIdx;
				_utfMsgTextTempThird := "";
				_utfMsgTextTempThird := DINT_TO_WSTRING(_MsgImage[_wImageIdx].diMsgAttr1);
			ELSE
				_utfMsgTextTempThird := "{##AttrVar1}";
			END_IF;
			_utfMsgTextTempSecond := "";
			_fbMsgReplSubStr.utfStr := ADR(_MsgTxtLine[_wTxtIdx].utfText);
			_fbMsgReplSubStr.utfSubStr := ADR("{##AttrVar1}");
			_fbMsgReplSubStr.utfStrToReplWith := ADR(_utfMsgTextTempThird);
			_fbMsgReplSubStr.utfStrResult := ADR(_utfMsgTextTempSecond);
			_fbMsgReplSubStr();
			IF _BinSearchCfg.wStatus = ERR_OK THEN
				_wImageIdx := _BinSearchCfg.wMsgIdx;
				_utfMsgTextTempThird := "";
				_utfMsgTextTempThird := DINT_TO_WSTRING(_MsgImage[_wImageIdx].diMsgAttr2);
			ELSE
				_utfMsgTextTempThird := "{##AttrVar2}";
			END_IF;
			_utfMsgTextTempFourth := "";
			_utfMsgTextTempFourth := _utfMsgTextTempSecond;
			_utfMsgTextTempSecond := "";
			_fbMsgReplSubStr.utfStr := ADR(_utfMsgTextTempFourth);
			_fbMsgReplSubStr.utfSubStr := ADR("{##AttrVar2}");
			_fbMsgReplSubStr.utfStrToReplWith := ADR(_utfMsgTextTempThird);
			_fbMsgReplSubStr.utfStrResult := ADR(_utfMsgTextTempSecond);
			_fbMsgReplSubStr();
			IF _BinSearchCfg.wStatus = ERR_OK THEN
				_wImageIdx := _BinSearchCfg.wMsgIdx;
				_utfMsgTextTempThird := "";
				_utfMsgTextTempThird := STRING_TO_WSTRING(_MsgImage[_wImageIdx].sMsgAttrTxt);
			ELSE
				_utfMsgTextTempThird := "{##AttrTxt}";
			END_IF;
			_utfMsgTextTempFourth := "";
			_utfMsgTextTempFourth := _utfMsgTextTempSecond;
			_utfMsgTextTempSecond := "";
			_fbMsgReplSubStr.utfStr := ADR(_utfMsgTextTempFourth);
			_fbMsgReplSubStr.utfSubStr := ADR("{##AttrTxt}");
			_fbMsgReplSubStr.utfStrToReplWith := ADR(_utfMsgTextTempThird);
			_fbMsgReplSubStr.utfStrResult := ADR(_utfMsgTextTempSecond);
			_fbMsgReplSubStr();
			brwcsncat(ADR(_utfMsgTextTempFirst), ADR(_utfMsgTextTempSecond),
			UDINT_TO_UINT(brwcslen(ADR(_utfMsgTextTempSecond)) - (brwcslen(ADR(_utfMsgTextTempFirst)) + brwcslen(ADR(_utfMsgTextTempSecond)) - (SIZEOF(_utfMsgTextTempFirst) / 2 - 1))));
			_utfMsgTextTempSecond := "";
			_utfMsgTextTempSecond := ": ";
			brwcsncat(ADR(_utfMsgTextTempFirst), ADR(_utfMsgTextTempSecond),
			UDINT_TO_UINT(brwcslen(ADR(_utfMsgTextTempSecond)) - (brwcslen(ADR(_utfMsgTextTempFirst)) + brwcslen(ADR(_utfMsgTextTempSecond)) - (SIZEOF(_utfMsgTextTempFirst) / 2 - 1))));
		END_IF;
		_MsgTxtLine ACCESS IFmnTxt.Out.ptrMessageTxtList;
		_BinSearchTxt.MsgTxtList := IFmnTxt.Out.ptrMessageTxtList;
		_BinSearchTxt.wCntMsgTxt := IFmnTxt.Out.wCntMessageTxt;
		_BinSearchTxt.wFunctionID := _wActFunctionID;
		_BinSearchTxt.wNumber := _wActMsgNumber;
		_BinSearchTxt.wInstance := _wActInstance;
		_BinSearchTxt.bTupel := 2;
		_BinSearchTxt();
		IF _BinSearchTxt.wStatus <> ERR_OK THEN
			brwcscat(ADR(_utfMsgTextTempFirst), ADR(""));
		ELSE
			_wTxtIdx := _BinSearchTxt.wMsgPos;
			_BinSearchCfg.wFunctionID := _wActFunctionID;
			_BinSearchCfg.wMsgNo := _wActMsgNumber;
			_BinSearchCfg.wInstance := _wActInstance;
			_BinSearchCfg();
			IF _BinSearchCfg.wStatus = ERR_OK THEN
				_wImageIdx := _BinSearchCfg.wMsgIdx;
				_utfMsgTextTempThird := "";
				_utfMsgTextTempThird := DINT_TO_WSTRING(_MsgImage[_wImageIdx].diMsgAttr1);
			ELSE
				_utfMsgTextTempThird := "{##AttrVar1}";
			END_IF;
			_utfMsgTextTempSecond := "";
			_fbMsgReplSubStr.utfStr := ADR(_MsgTxtLine[_wTxtIdx].utfText);
			_fbMsgReplSubStr.utfSubStr := ADR("{##AttrVar1}");
			_fbMsgReplSubStr.utfStrToReplWith := ADR(_utfMsgTextTempThird);
			_fbMsgReplSubStr.utfStrResult := ADR(_utfMsgTextTempSecond);
			_fbMsgReplSubStr();
			IF _BinSearchCfg.wStatus = ERR_OK THEN
				_wImageIdx := _BinSearchCfg.wMsgIdx;
				_utfMsgTextTempThird := "";
				_utfMsgTextTempThird := DINT_TO_WSTRING(_MsgImage[_wImageIdx].diMsgAttr2);
			ELSE
				_utfMsgTextTempThird := "{##AttrVar2}";
			END_IF;
			_utfMsgTextTempFourth := "";
			_utfMsgTextTempFourth := _utfMsgTextTempSecond;
			_utfMsgTextTempSecond := "";
			_fbMsgReplSubStr.utfStr := ADR(_utfMsgTextTempFourth);
			_fbMsgReplSubStr.utfSubStr := ADR("{##AttrVar2}");
			_fbMsgReplSubStr.utfStrToReplWith := ADR(_utfMsgTextTempThird);
			_fbMsgReplSubStr.utfStrResult := ADR(_utfMsgTextTempSecond);
			_fbMsgReplSubStr();
			IF _BinSearchCfg.wStatus = ERR_OK THEN
				_wImageIdx := _BinSearchCfg.wMsgIdx;
				_utfMsgTextTempThird := "";
				_utfMsgTextTempThird := STRING_TO_WSTRING(_MsgImage[_wImageIdx].sMsgAttrTxt);
			ELSE
				_utfMsgTextTempThird := "{##AttrTxt}";
			END_IF;
			_utfMsgTextTempFourth := "";
			_utfMsgTextTempFourth := _utfMsgTextTempSecond;
			_utfMsgTextTempSecond := "";
			_fbMsgReplSubStr.utfStr := ADR(_utfMsgTextTempFourth);
			_fbMsgReplSubStr.utfSubStr := ADR("{##AttrTxt}");
			_fbMsgReplSubStr.utfStrToReplWith := ADR(_utfMsgTextTempThird);
			_fbMsgReplSubStr.utfStrResult := ADR(_utfMsgTextTempSecond);
			_fbMsgReplSubStr();
			brwcsncat(ADR(_utfMsgTextTempFirst), ADR(_utfMsgTextTempSecond),
			UDINT_TO_UINT(brwcslen(ADR(_utfMsgTextTempSecond)) - (brwcslen(ADR(_utfMsgTextTempFirst)) + brwcslen(ADR(_utfMsgTextTempSecond)) - (SIZEOF(_utfMsgTextTempFirst) / 2 - 1))));
		END_IF;
	ELSE
		brwcscat(ADR(_utfMsgTextTempFirst), ADR(""));
	END_IF;
END_ACTION
```

#### _actGetTxtFimh.st
```iecst
(********************************************************************
 * COPYRIGHT -- Herbert Kannegiesser GmbH
 ********************************************************************
 * Program: mnMsg
 * File: actGetTxtFimh.st
 * Author: kuehne
 * Created: February 22, 2012
 ********************************************************************
 * Implementation of program mnMsg
 ********************************************************************)

 (* Add a new action to your IEC program or library *)
ACTION _actGetTxtFimh:
	IF _xMnTxtReady THEN
		_MsgTxtLine ACCESS IFmnTxt.Out.ptrFunctionTxtList;
		_BinSearchTxt.MsgTxtList := IFmnTxt.Out.ptrFunctionTxtList;
		_BinSearchTxt.wCntMsgTxt := IFmnTxt.Out.wCntFunctionTxt;
		_BinSearchTxt.wFunctionID := _wActFunctionID;
		_BinSearchTxt.wNumber := _wActMsgNumber;
		_BinSearchTxt.wInstance := _wActInstance;
		_BinSearchTxt.bTupel := 1;
		_BinSearchTxt();
		IF _BinSearchTxt.wStatus <> ERR_OK THEN
			brwcscat(ADR(_utfMsgTextTempFirst), ADR(""));
		ELSE
			_wTxtIdx := _BinSearchTxt.wMsgPos;
			_utfMsgTextTempSecond := "";
			_utfMsgTextTempThird := "";
			_utfMsgTextTempThird := DINT_TO_WSTRING(_diActAttr1);
			_fbMsgReplSubStr.utfStr := ADR(_MsgTxtLine[_wTxtIdx].utfText);
			_fbMsgReplSubStr.utfSubStr := ADR("{##AttrVar1}");
			_fbMsgReplSubStr.utfStrToReplWith := ADR(_utfMsgTextTempThird);
			_fbMsgReplSubStr.utfStrResult := ADR(_utfMsgTextTempSecond);
			_fbMsgReplSubStr();
			_utfMsgTextTempThird := "";
			_utfMsgTextTempFourth := "";
			_utfMsgTextTempFourth := _utfMsgTextTempSecond;
			_utfMsgTextTempSecond := "";
			_utfMsgTextTempThird := DINT_TO_WSTRING(_diActAttr2);
			_fbMsgReplSubStr.utfStr := ADR(_utfMsgTextTempFourth);
			_fbMsgReplSubStr.utfSubStr := ADR("{##AttrVar2}");
			_fbMsgReplSubStr.utfStrToReplWith := ADR(_utfMsgTextTempThird);
			_fbMsgReplSubStr.utfStrResult := ADR(_utfMsgTextTempSecond);
			_fbMsgReplSubStr();
			_utfMsgTextTempThird := "";
			_utfMsgTextTempFourth := "";
			_utfMsgTextTempFourth := _utfMsgTextTempSecond;
			_utfMsgTextTempSecond := "";
			_utfMsgTextTempThird := STRING_TO_WSTRING(_sActAttrTxt);
			_fbMsgReplSubStr.utfStr := ADR(_utfMsgTextTempFourth);
			_fbMsgReplSubStr.utfSubStr := ADR("{##AttrTxt}");
			_fbMsgReplSubStr.utfStrToReplWith := ADR(_utfMsgTextTempThird);
			_fbMsgReplSubStr.utfStrResult := ADR(_utfMsgTextTempSecond);
			_fbMsgReplSubStr();
			brwcsncat(ADR(_utfMsgTextTempFirst), ADR(_utfMsgTextTempSecond),
			UDINT_TO_UINT(brwcslen(ADR(_utfMsgTextTempSecond)) - (brwcslen(ADR(_utfMsgTextTempFirst)) + brwcslen(ADR(_utfMsgTextTempSecond)) - (SIZEOF(_utfMsgTextTempFirst) / 2 - 1))));
			_utfMsgTextTempSecond := ": ";
			brwcsncat(ADR(_utfMsgTextTempFirst), ADR(_utfMsgTextTempSecond),
			UDINT_TO_UINT(brwcslen(ADR(_utfMsgTextTempSecond)) - (brwcslen(ADR(_utfMsgTextTempFirst)) + brwcslen(ADR(_utfMsgTextTempSecond)) - (SIZEOF(_utfMsgTextTempFirst) / 2 - 1))));
		END_IF;
		_MsgTxtLine ACCESS IFmnTxt.Out.ptrInstanceTxtList;
		_BinSearchTxt.MsgTxtList := IFmnTxt.Out.ptrInstanceTxtList;
		_BinSearchTxt.wCntMsgTxt := IFmnTxt.Out.wCntInstanceTxt;
		_BinSearchTxt.wFunctionID := _wActFunctionID;
		_BinSearchTxt.wNumber := _wActInstance;
		_BinSearchTxt.wInstance := 0;
		_BinSearchTxt.bTupel := 2;
		_BinSearchTxt();
		IF _BinSearchTxt.wStatus <> ERR_OK THEN
			brwcscat(ADR(_utfMsgTextTempFirst), ADR(""));
		ELSE
			_wTxtIdx := _BinSearchTxt.wMsgPos;
			_utfMsgTextTempSecond := "";
			_utfMsgTextTempThird := "";
			_utfMsgTextTempThird := DINT_TO_WSTRING(_diActAttr1);
			_fbMsgReplSubStr.utfStr := ADR(_MsgTxtLine[_wTxtIdx].utfText);
			_fbMsgReplSubStr.utfSubStr := ADR("{##AttrVar1}");
			_fbMsgReplSubStr.utfStrToReplWith := ADR(_utfMsgTextTempThird);
			_fbMsgReplSubStr.utfStrResult := ADR(_utfMsgTextTempSecond);
			_fbMsgReplSubStr();
			_utfMsgTextTempThird := "";
			_utfMsgTextTempFourth := "";
			_utfMsgTextTempFourth := _utfMsgTextTempSecond;
			_utfMsgTextTempSecond := "";
			_utfMsgTextTempThird := DINT_TO_WSTRING(_diActAttr2);
			_fbMsgReplSubStr.utfStr := ADR(_utfMsgTextTempFourth);
			_fbMsgReplSubStr.utfSubStr := ADR("{##AttrVar2}");
			_fbMsgReplSubStr.utfStrToReplWith := ADR(_utfMsgTextTempThird);
			_fbMsgReplSubStr.utfStrResult := ADR(_utfMsgTextTempSecond);
			_fbMsgReplSubStr();
			_utfMsgTextTempThird := "";
			_utfMsgTextTempFourth := "";
			_utfMsgTextTempFourth := _utfMsgTextTempSecond;
			_utfMsgTextTempSecond := "";
			_utfMsgTextTempThird := STRING_TO_WSTRING(_sActAttrTxt);
			_fbMsgReplSubStr.utfStr := ADR(_utfMsgTextTempFourth);
			_fbMsgReplSubStr.utfSubStr := ADR("{##AttrTxt}");
			_fbMsgReplSubStr.utfStrToReplWith := ADR(_utfMsgTextTempThird);
			_fbMsgReplSubStr.utfStrResult := ADR(_utfMsgTextTempSecond);
			_fbMsgReplSubStr();
			brwcsncat(ADR(_utfMsgTextTempFirst), ADR(_utfMsgTextTempSecond),
			UDINT_TO_UINT(brwcslen(ADR(_utfMsgTextTempSecond)) - (brwcslen(ADR(_utfMsgTextTempFirst)) + brwcslen(ADR(_utfMsgTextTempSecond)) - (SIZEOF(_utfMsgTextTempFirst) / 2 - 1))));
			_utfMsgTextTempSecond := "";
			_utfMsgTextTempSecond := ": ";
			brwcsncat(ADR(_utfMsgTextTempFirst), ADR(_utfMsgTextTempSecond),
			UDINT_TO_UINT(brwcslen(ADR(_utfMsgTextTempSecond)) - (brwcslen(ADR(_utfMsgTextTempFirst)) + brwcslen(ADR(_utfMsgTextTempSecond)) - (SIZEOF(_utfMsgTextTempFirst) / 2 - 1))));
		END_IF;
		_MsgTxtLine ACCESS IFmnTxt.Out.ptrMessageTxtList;
		_BinSearchTxt.MsgTxtList := IFmnTxt.Out.ptrMessageTxtList;
		_BinSearchTxt.wCntMsgTxt := IFmnTxt.Out.wCntMessageTxt;
		_BinSearchTxt.wFunctionID := _wActFunctionID;
		_BinSearchTxt.wNumber := _wActMsgNumber;
		_BinSearchTxt.wInstance := _wActInstance;
		_BinSearchTxt.bTupel := 2;
		_BinSearchTxt();
		IF _BinSearchTxt.wStatus <> ERR_OK THEN
			brwcscat(ADR(_utfMsgTextTempFirst), ADR(""));
		ELSE
			_wTxtIdx := _BinSearchTxt.wMsgPos;
			_utfMsgTextTempSecond := "";
			_utfMsgTextTempThird := "";
			_utfMsgTextTempThird := DINT_TO_WSTRING(_diActAttr1);
			_fbMsgReplSubStr.utfStr := ADR(_MsgTxtLine[_wTxtIdx].utfText);
			_fbMsgReplSubStr.utfSubStr := ADR("{##AttrVar1}");
			_fbMsgReplSubStr.utfStrToReplWith := ADR(_utfMsgTextTempThird);
			_fbMsgReplSubStr.utfStrResult := ADR(_utfMsgTextTempSecond);
			_fbMsgReplSubStr();
			_utfMsgTextTempThird := "";
			_utfMsgTextTempFourth := "";
			_utfMsgTextTempFourth := _utfMsgTextTempSecond;
			_utfMsgTextTempSecond := "";
			_utfMsgTextTempThird := DINT_TO_WSTRING(_diActAttr2);
			_fbMsgReplSubStr.utfStr := ADR(_utfMsgTextTempFourth);
			_fbMsgReplSubStr.utfSubStr := ADR("{##AttrVar2}");
			_fbMsgReplSubStr.utfStrToReplWith := ADR(_utfMsgTextTempThird);
			_fbMsgReplSubStr.utfStrResult := ADR(_utfMsgTextTempSecond);
			_fbMsgReplSubStr();
			_utfMsgTextTempThird := "";
			_utfMsgTextTempFourth := "";
			_utfMsgTextTempFourth := _utfMsgTextTempSecond;
			_utfMsgTextTempSecond := "";
			_utfMsgTextTempThird := STRING_TO_WSTRING(_sActAttrTxt);
			_fbMsgReplSubStr.utfStr := ADR(_utfMsgTextTempFourth);
			_fbMsgReplSubStr.utfSubStr := ADR("{##AttrTxt}");
			_fbMsgReplSubStr.utfStrToReplWith := ADR(_utfMsgTextTempThird);
			_fbMsgReplSubStr.utfStrResult := ADR(_utfMsgTextTempSecond);
			_fbMsgReplSubStr();
			brwcsncat(ADR(_utfMsgTextTempFirst), ADR(_utfMsgTextTempSecond),
			UDINT_TO_UINT(brwcslen(ADR(_utfMsgTextTempSecond)) - (brwcslen(ADR(_utfMsgTextTempFirst)) + brwcslen(ADR(_utfMsgTextTempSecond)) - (SIZEOF(_utfMsgTextTempFirst) / 2 - 1))));
		END_IF;
		// wcscat(ADR(_utfMsgTextTempFirst), ADR("internal error"));	//Also for test
		_MsgHelpTxtLine ACCESS IFmnTxt.Out.ptrMessageHelpTxtList;
		_BinSearchHelpTxt.MsgHelpTxtList := IFmnTxt.Out.ptrMessageHelpTxtList;
		_BinSearchHelpTxt.wCntMsgHelpTxt := IFmnTxt.Out.wCntMessageHlpTxt;
		_BinSearchHelpTxt.wFunctionID := _wActFunctionID;
		_BinSearchHelpTxt.wNumber := _wActMsgNumber;
		_BinSearchHelpTxt.wInstance := _wActInstance;
		_BinSearchHelpTxt.bTupel := 2;
		_BinSearchHelpTxt();
		IF _BinSearchHelpTxt.wStatus <> ERR_OK THEN
			_utfMsgTextTempSecond := "";
		ELSE
			_wTxtIdx := _BinSearchHelpTxt.wMsgPos;
			_utfMsgTextTempSecond := "";
			_utfMsgTextTempThird := "";
			_utfMsgTextTempThird := DINT_TO_WSTRING(_diActAttr1);
			_fbMsgReplSubStr.utfStr := ADR(_MsgHelpTxtLine[_wTxtIdx].utfText);
			_fbMsgReplSubStr.utfSubStr := ADR("{##AttrVar1}");
			_fbMsgReplSubStr.utfStrToReplWith := ADR(_utfMsgTextTempThird);
			_fbMsgReplSubStr.utfStrResult := ADR(_utfMsgTextTempSecond);
			_fbMsgReplSubStr();
			_utfMsgTextTempThird := "";
			_utfMsgTextTempFourth := "";
			_utfMsgTextTempFourth := _utfMsgTextTempSecond;
			_utfMsgTextTempSecond := "";
			_utfMsgTextTempThird := DINT_TO_WSTRING(_diActAttr2);
			_fbMsgReplSubStr.utfStr := ADR(_utfMsgTextTempFourth);
			_fbMsgReplSubStr.utfSubStr := ADR("{##AttrVar2}");
			_fbMsgReplSubStr.utfStrToReplWith := ADR(_utfMsgTextTempThird);
			_fbMsgReplSubStr.utfStrResult := ADR(_utfMsgTextTempSecond);
			_fbMsgReplSubStr();
			_utfMsgTextTempThird := "";
			_utfMsgTextTempFourth := "";
			_utfMsgTextTempFourth := _utfMsgTextTempSecond;
			_utfMsgTextTempSecond := "";
			_utfMsgTextTempThird := STRING_TO_WSTRING(_sActAttrTxt);
			_fbMsgReplSubStr.utfStr := ADR(_utfMsgTextTempFourth);
			_fbMsgReplSubStr.utfSubStr := ADR("{##AttrTxt}");
			_fbMsgReplSubStr.utfStrToReplWith := ADR(_utfMsgTextTempThird);
			_fbMsgReplSubStr.utfStrResult := ADR(_utfMsgTextTempSecond);
			_fbMsgReplSubStr();
		END_IF;
	ELSE
		brwcscat(ADR(_utfMsgTextTempFirst), ADR(""));
		brwcscat(ADR(_utfMsgTextTempSecond), ADR(""));
	END_IF; // IF _xMnTxtReady THEN
END_ACTION
```

#### _actGetOneTurnRB.st
```iecst
(********************************************************************
 * COPYRIGHT -- Herbert Kannegiesser GmbH
 ********************************************************************
 * Program: mnMsg
 * File: actGetOneTurnRB.st
 * Author: kuehne
 * Created: February 22, 2012
 ********************************************************************
 * Implementation of program mnMsg
 ********************************************************************)

(* Add a new action to your IEC program or library *)
ACTION _actGetOneTurnRB:
	IF _xRBReady THEN
		IF _wPtrRBstart = 0 THEN
			_xRBoneTurn := FALSE;
			IF _wPtrRBwrite > 0 THEN
				_wMsgHistListMaxOffsetRB := _wPtrRBwrite - 1;
			ELSE
				_wMsgHistListMaxOffsetRB := 0;
			END_IF;
		END_IF;
		IF _wPtrRBstart = _wPtrRBwrite + 1 THEN
			_xRBoneTurn := TRUE;
			_wMsgHistListMaxOffsetRB := MNMSG_MAX_MESSAGEHISTORY - 1;
		END_IF;
	ELSE
		_xRBoneTurn := FALSE;
		_wMsgHistListMaxOffsetRB := 0;
	END_IF;
END_ACTION
```

#### _actSetMsgOrMaint.st
```iecst
(********************************************************************
 * COPYRIGHT -- Herbert Kannegiesser GmbH
 ********************************************************************
 * Program: mnMsg
 * File: actSetMsgOrMaint.st
 * Author: kuehne
 * Created: February 22, 2012
 ********************************************************************
 * Implementation of program mnMsg
 ********************************************************************)

 (* Add a new action to your IEC program or library *)
ACTION _actSetMsgOrMaint:
	IF kgMsgStatus[_wSrcIdx].wMsgClass = 20 THEN
		IF kgMsgStatus[_wSrcIdx].wMaintNumber = 0 AND kgMsgStatus[_wSrcIdx].wMsgNumber <> 0 THEN
			kgMsgStatus[_wSrcIdx].wMaintNumber := kgMsgStatus[_wSrcIdx].wMsgNumber;
		END_IF;
		kgMsgStatus[_wSrcIdx].wMsgNumber := 0;
		IF kgMsgStatus[_wSrcIdx].wMaintAckLevel = 0 AND kgMsgStatus[_wSrcIdx].wMsgAckLevel <> 0 THEN
			kgMsgStatus[_wSrcIdx].wMaintAckLevel := kgMsgStatus[_wSrcIdx].wMsgAckLevel;
		END_IF;
		kgMsgStatus[_wSrcIdx].wMsgAckLevel := 0;
		IF kgMsgStatus[_wSrcIdx].diMaintAttr1 = 0 AND kgMsgStatus[_wSrcIdx].diMsgAttr1 <> 0 THEN
			kgMsgStatus[_wSrcIdx].diMaintAttr1 := kgMsgStatus[_wSrcIdx].diMsgAttr1;
		END_IF;
		kgMsgStatus[_wSrcIdx].diMsgAttr1 := 0;
		IF kgMsgStatus[_wSrcIdx].diMaintAttr2 = 0 AND kgMsgStatus[_wSrcIdx].diMsgAttr2 <> 0 THEN
			kgMsgStatus[_wSrcIdx].diMaintAttr2 := kgMsgStatus[_wSrcIdx].diMsgAttr2;
		END_IF;
		kgMsgStatus[_wSrcIdx].diMsgAttr2 := 0;
		IF kgMsgStatus[_wSrcIdx].sMaintAttrTxt = '' AND kgMsgStatus[_wSrcIdx].sMsgAttrTxt <> '' THEN
			kgMsgStatus[_wSrcIdx].sMaintAttrTxt := kgMsgStatus[_wSrcIdx].sMsgAttrTxt;
		END_IF;
		kgMsgStatus[_wSrcIdx].sMsgAttrTxt := '';
	END_IF;
	IF kgMsgStatus[_wSrcIdx].wMsgClass = 0 OR kgMsgStatus[_wSrcIdx].wMsgClass = 1 OR kgMsgStatus[_wSrcIdx].wMsgClass = 10 OR kgMsgStatus[_wSrcIdx].wMsgClass = 11 THEN
		IF kgMsgStatus[_wSrcIdx].wMsgNumber = 0 AND kgMsgStatus[_wSrcIdx].wMaintNumber <> 0 THEN
			kgMsgStatus[_wSrcIdx].wMsgNumber := kgMsgStatus[_wSrcIdx].wMaintNumber;
		END_IF;
		kgMsgStatus[_wSrcIdx].wMaintNumber := 0;
		IF kgMsgStatus[_wSrcIdx].wMsgAckLevel = 0 AND kgMsgStatus[_wSrcIdx].wMaintAckLevel <> 0 THEN
			kgMsgStatus[_wSrcIdx].wMsgAckLevel := kgMsgStatus[_wSrcIdx].wMaintAckLevel;
		END_IF;
		kgMsgStatus[_wSrcIdx].wMaintAckLevel := 0;
		IF kgMsgStatus[_wSrcIdx].diMsgAttr1 = 0 AND kgMsgStatus[_wSrcIdx].diMaintAttr1 <> 0 THEN
			kgMsgStatus[_wSrcIdx].diMsgAttr1 := kgMsgStatus[_wSrcIdx].diMaintAttr1;
		END_IF;
		kgMsgStatus[_wSrcIdx].diMaintAttr1 := 0;
		IF kgMsgStatus[_wSrcIdx].diMsgAttr2 = 0 AND kgMsgStatus[_wSrcIdx].diMaintAttr2 <> 0 THEN
			kgMsgStatus[_wSrcIdx].diMsgAttr2 := kgMsgStatus[_wSrcIdx].diMaintAttr2;
		END_IF;
		kgMsgStatus[_wSrcIdx].diMaintAttr2 := 0;
		IF kgMsgStatus[_wSrcIdx].sMsgAttrTxt = '' AND kgMsgStatus[_wSrcIdx].sMaintAttrTxt <> '' THEN
			kgMsgStatus[_wSrcIdx].sMsgAttrTxt := kgMsgStatus[_wSrcIdx].sMaintAttrTxt;
		END_IF;
		kgMsgStatus[_wSrcIdx].sMaintAttrTxt := '';
	END_IF;
END_ACTION
```

#### _actInsertRB.st
```iecst
(********************************************************************
 * COPYRIGHT -- Herbert Kannegiesser GmbH
 ********************************************************************
 * Program: mnMsg
 * File: actInsertRB.st
 * Author: kuehne
 * Created: February 22, 2012
 ********************************************************************
 * Implementation of program mnMsg
 ********************************************************************)

(* Add a new action to your IEC program or library *)
ACTION _actInsertRB:
	IF _xRBReady THEN
		_TempHistline.TimeStampEvent := _dtTimeStamp.DT1;
		_TempHistline.wFunction_ID := _MsgCfgList[_wMsgIdx].wFunction_ID;
		_TempHistline.wInstance := _MsgCfgList[_wMsgIdx].wInstance;
		_TempHistline.wMsgNumber := _MsgCfgList[_wMsgIdx].wMsgNumber;
		_TempHistline.wMsgClass := _MsgImage[_wMsgIdx].wMsgClass;
		_TempHistline.diAttr1 := _MsgImage[_wMsgIdx].diMsgAttr1;
		_TempHistline.diAttr2 := _MsgImage[_wMsgIdx].diMsgAttr2;
		strcpy(ADR(_TempHistline.sAttrTxt), ADR(_MsgImage[_wMsgIdx].sMsgAttrTxt));
		_TempHistline.lTime := _lActTime;
		_TempHistline.wEvent := _wActEvent;
		_InsertRB(wPtrWrite := _wPtrRBwrite, wPtrRead := _wPtrRBread, wPtrStart := _wPtrRBstart);
	END_IF;
END_ACTION
```

#### _actInsertMsgL.st
```iecst
(********************************************************************
 * COPYRIGHT -- Herbert Kannegiesser GmbH
 ********************************************************************
 * Program: mnMsg
 * File: actInsertMsgL.st
 * Author: kuehne
 * Created: February 23, 2012
 ********************************************************************
 * Implementation of program mnMsg
 ********************************************************************)

(* Add a new action to your IEC program or library *)
ACTION _actInsertMsgL:
	_InsertMsgLine.Class := _bActMsgLClass;
	_InsertMsgLine.Insert := TRUE;
	_InsertMsgLine.MsgLine.wFunction_ID :=  _MsgCfgList[_wMsgIdx].wFunction_ID;
	_InsertMsgLine.MsgLine.wMsgNumber := _MsgCfgList[_wMsgIdx].wMsgNumber;
	_InsertMsgLine.MsgLine.bInstance := UINT_TO_USINT(_MsgCfgList[_wMsgIdx].wInstance);
	_InsertMsgLine.MsgLine.bAckLevel := UINT_TO_USINT(_MsgImage[_wMsgIdx].wMsgAckLevel);
	_InsertMsgLine.MsgLine.TimeStamp := _MsgImageTime[_wMsgIdx].dtTimeStamp;
	_InsertMsgLine.MsgLine.diAttr1 := _MsgImage[_wMsgIdx].diMsgAttr1;
	_InsertMsgLine.MsgLine.diAttr2 := _MsgImage[_wMsgIdx].diMsgAttr2;
	strcpy(ADR(_InsertMsgLine.MsgLine.sAttrTxt),ADR(_MsgImage[_wMsgIdx].sMsgAttrTxt));
	_InsertMsgLine();
END_ACTION
```

#### _actStatisticTextLCID.st
```iecst
(********************************************************************
 * COPYRIGHT -- Herbert Kannegiesser GmbH
 ********************************************************************
 * Program: mnMsg
 * File: actStatisticTextLCID.st
 * Author: kuehne
 * Created: February 24, 2012
 ********************************************************************
 * Implementation of program mnMsg
 ********************************************************************)

(* Add a new action to your IEC program or library *)
ACTION _actStatisticTextLCID:
	_GetNextChrPos.lStartPos := 0;
	_GetNextChrPos.utfStr := ADR(_utfMsgTxtLCIDfirst);
	_GetNextChrPos.utfChr := ".";
	_GetNextChrPos();
	_lPosPointFirst := _GetNextChrPos.lChrPos;
	_lAdrPointFirst := ADR(_utfMsgTxtLCIDfirst) + 2 * _lPosPointFirst;
	//
	_GetNextChrPos.lStartPos := _lPosPointFirst + 1;
	_GetNextChrPos.utfStr := ADR(_utfMsgTxtLCIDfirst);
	_GetNextChrPos.utfChr := ".";
	_GetNextChrPos();
	_lPosPointSecond := _GetNextChrPos.lChrPos;
	_lAdrPointSecond := ADR(_utfMsgTxtLCIDfirst) + 2 * _lPosPointSecond;
	//
	_GetNextChrPos.lStartPos := _lPosPointSecond + 1;
	_GetNextChrPos.utfStr := ADR(_utfMsgTxtLCIDfirst);
	_GetNextChrPos.utfChr := " ";
	_GetNextChrPos();
	_lPosSpaceFirst := _GetNextChrPos.lChrPos;
	_lAdrSpaceFirst := ADR(_utfMsgTxtLCIDfirst) + 2 * _lPosSpaceFirst;
	//
	IF (_lPosPointFirst > 0) AND (_lPosPointFirst < (SIZEOF(_utfLCIDFunctionId) / 2)) THEN
		_utfLCIDFunctionId := "";
		wcsncat(ADR(_utfLCIDFunctionId), ADR(_utfMsgTxtLCIDfirst), _lPosPointFirst);
		_wLCIDFunctionId := WSTRING_TO_UINT(_utfLCIDFunctionId);
	ELSE
		_utfLCIDFunctionId := "";
		_wLCIDFunctionId := 0;
	END_IF;
	IF ((_lPosPointSecond - 1 - _lPosPointFirst) > 0) AND ((_lPosPointSecond - 1 - _lPosPointFirst) < (SIZEOF(_utfLCIDMsgNumber) / 2)) THEN
		_utfLCIDMsgNumber := "";
		wcsncat(ADR(_utfLCIDMsgNumber), _lAdrPointFirst + 2, _lPosPointSecond - 1 - _lPosPointFirst);
		_wLCIDMsgNumber := WSTRING_TO_UINT(_utfLCIDMsgNumber);
	ELSE
		_utfLCIDMsgNumber := "";
		_wLCIDMsgNumber := 0;
	END_IF;
	IF ((_lPosSpaceFirst - 1 - _lPosPointSecond) > 0) AND ((_lPosSpaceFirst - 1 - _lPosPointSecond) < (SIZEOF(_utfLCIDInstance) / 2)) THEN
		_utfLCIDInstance := "";
		wcsncat(ADR(_utfLCIDInstance), _lAdrPointSecond + 2, _lPosSpaceFirst - 1 - _lPosPointSecond);
		_wLCIDInstance := WSTRING_TO_UINT(_utfLCIDInstance);
	ELSE
		_utfLCIDInstance := "";
		_wLCIDInstance := 0;
	END_IF;
	_utfMsgTxtLCIDfirst := "";
	wcsncat(ADR(_utfMsgTxtLCIDfirst), ADR(_utfLCIDFunctionId),
	UDINT_TO_UINT(wcslen(ADR(_utfLCIDFunctionId)) - (wcslen(ADR(_utfMsgTxtLCIDfirst)) + wcslen(ADR(_utfLCIDFunctionId)) - (SIZEOF(_utfMsgTxtLCIDfirst) / 2 - 1))));
	wcsncat(ADR(_utfMsgTxtLCIDfirst), ADR("."),
	UDINT_TO_UINT(wcslen(ADR(".")) - (wcslen(ADR(_utfMsgTxtLCIDfirst)) + wcslen(ADR(".")) - (SIZEOF(_utfMsgTxtLCIDfirst) / 2 - 1))));
	wcsncat(ADR(_utfMsgTxtLCIDfirst), ADR(_utfLCIDMsgNumber),
	UDINT_TO_UINT(wcslen(ADR(_utfLCIDMsgNumber)) - (wcslen(ADR(_utfMsgTxtLCIDfirst)) + wcslen(ADR(_utfLCIDMsgNumber)) - (SIZEOF(_utfMsgTxtLCIDfirst) / 2 - 1))));
	wcsncat(ADR(_utfMsgTxtLCIDfirst), ADR("."),
	UDINT_TO_UINT(wcslen(ADR(".")) - (wcslen(ADR(_utfMsgTxtLCIDfirst)) + wcslen(ADR(".")) - (SIZEOF(_utfMsgTxtLCIDfirst) / 2 - 1))));
	wcsncat(ADR(_utfMsgTxtLCIDfirst), ADR(_utfLCIDInstance),
	UDINT_TO_UINT(wcslen(ADR(_utfLCIDInstance)) - (wcslen(ADR(_utfMsgTxtLCIDfirst)) + wcslen(ADR(_utfLCIDInstance)) - (SIZEOF(_utfMsgTxtLCIDfirst) / 2 - 1))));
	wcsncat(ADR(_utfMsgTxtLCIDfirst), ADR(" "),
	UDINT_TO_UINT(wcslen(ADR(" ")) - (wcslen(ADR(_utfMsgTxtLCIDfirst)) + wcslen(ADR(" ")) - (SIZEOF(_utfMsgTxtLCIDfirst) / 2 - 1))));
	_wActFunctionID := _wLCIDFunctionId;
	_wActMsgNumber := _wLCIDMsgNumber;
	_wActInstance := _wLCIDInstance;
	_utfMsgTextTempFirst := "";
	_utfMsgTextTempFirst := _utfMsgTxtLCIDfirst;
	_actGetTxtFim;
	_utfMsgTxtLCIDfirst := "";
	_utfMsgTxtLCIDfirst := _utfMsgTextTempFirst;
END_ACTION
```

#### _actLocMOD.st
```iecst
(********************************************************************
 * COPYRIGHT -- Herbert Kannegiesser GmbH
 ********************************************************************
 * Program: mnMsg
 * File: actLocMOD.st
 * Author: kuehne
 * Created: February 24, 2012
 ********************************************************************
 * Implementation of program mnMsg
 ********************************************************************)

(* Add a new action to your IEC program or library *)
ACTION _actLocMOD:
	IF _xRBoneTurn THEN
		IF MNMSG_MAX_MESSAGEHISTORY >= 1 AND (_wPtrRBloc + _wMsgHistListOffsetRB) > 0 THEN
			_wPtrRBloc := (_wPtrRBloc + _wMsgHistListOffsetRB) MOD UDINT_TO_UINT(MNMSG_MAX_MESSAGEHISTORY); // sum equals cnt: 0
		ELSE
			_wPtrRBloc := 0;
		END_IF;
	ELSE
		IF _wPtrRBwrite > 0 AND (_wPtrRBloc + _wMsgHistListOffsetRB) > 0 THEN
			_wPtrRBloc := (_wPtrRBloc + _wMsgHistListOffsetRB) MOD _wPtrRBwrite; // sum equals ptr: 0
		ELSE
			_wPtrRBloc := 0;
		END_IF;
	END_IF;
	IF _wPtrRBloc > _wPtrRBlocTemp THEN
		_wMsgHistListOffsetRB := _wPtrRBloc - _wPtrRBlocTemp;
	ELSE
		_wMsgHistListOffsetRB := 0;
	END_IF;
END_ACTION
```

#### _actEventClassSel.st
```iecst
(********************************************************************
 * COPYRIGHT -- Herbert Kannegiesser GmbH
 ********************************************************************
 * Program: mnMsg
 * File: actEventClassSel.st
 * Author: kuehne
 * Created: February 24, 2012
 ********************************************************************
 * Implementation of program mnMsg
 ********************************************************************)

(* Add a new action to your IEC program or library *)
ACTION _actEventClassSel:
	IF (_TempHistline.wEvent <> _wMsgHistListEventSelRB) AND (_wMsgHistListEventSelRB <> 0) THEN
		_xSelOk := FALSE;
	ELSIF ((_TempHistline.wMsgClass = 0) OR (_TempHistline.wMsgClass = 1)) AND (_wMsgHistListClassSelRB.0 = 0) THEN
		_xSelOk := FALSE;
	ELSIF (_TempHistline.wMsgClass = 10) AND (_wMsgHistListClassSelRB.1  = 0) THEN
		_xSelOk := FALSE;
	ELSIF (_TempHistline.wMsgClass = 11) AND (_wMsgHistListClassSelRB.2 = 0) THEN
		_xSelOk := FALSE;
	ELSIF (_TempHistline.wMsgClass = 20) AND (_wMsgHistListClassSelRB.3 = 0) THEN
		_xSelOk := FALSE;
	ELSE
		_wPtrRBlocLastFound := _wPtrRBloc;
		_xSelOk := TRUE;
	END_IF;
END_ACTION
```

### Library Logical/Standard/Kanlink/KGFramework/Pkg_mnMsg/KGlibMsg (IEC) - A new source library

#### KGlibMsg.typ - Exported data types
```iecst
(********************************************************************
 * COPYRIGHT -- Herbert Kannegiesser GmbH
 ********************************************************************
 * Library: KGlibMsg
 * File: KGlibMsg.typ
 * Author: hunholz
 * Created: May 30, 2011
 * Changed: June 15, 2011
 ********************************************************************
 * Data types of library KGlibMsg
 ********************************************************************)

TYPE
	MsgCfgLine_Typ : 	STRUCT
		wFunction_ID : UINT;
		wMsgNumber : UINT;
		wInstance : UINT;
		wRes : UINT;
	END_STRUCT;
	MsgHistList_Typ : 	STRUCT
		TimeStampEvent : DATE_AND_TIME;
		wFunction_ID : UINT;
		wMsgNumber : UINT;
		wInstance : UINT;
		wMsgClass : UINT;
		diAttr1 : DINT;
		diAttr2 : DINT;
		sAttrTxt : STRING[13];
		wEvent : UINT;
		lTime : UDINT;
	END_STRUCT;
	IFMsgHistList_Typ : 	STRUCT
		utfMsgText : WSTRING[67];
		bMsgClass : USINT;
		bEvent : USINT;
	END_STRUCT;
	MsgList_Typ : 	STRUCT
		TimeStamp : DATE_AND_TIME;
		wFunction_ID : UINT;
		wMsgNumber : UINT;
		bInstance : USINT;
		bAckLevel : USINT;
		sAttrTxt : STRING[13];
		diAttr1 : DINT;
		diAttr2 : DINT;
	END_STRUCT;
	MsgTxtLine_Typ : 	STRUCT
		wFunctionID : UINT;
		wNumber : UINT;
		wInstance : UINT;
		utfText : WSTRING[63];
	END_STRUCT;
	MsgHelpTxtLine_Typ : 	STRUCT
		wFunctionID : UINT;
		wNumber : UINT;
		wInstance : UINT;
		utfText : WSTRING[255];
	END_STRUCT;
	MsgKgMsgStatus_Typ : 	STRUCT
		wFunctionID : UINT;
		wMsgClass : UINT;
		wNumber : UINT;
		wMsgAckLevel : UINT;
		wInstance : UINT;
		sMsgAttrTxt : STRING[13];
		diMsgAttr1 : DINT;
		diMsgAttr2 : DINT;
		wMaintNumber : UINT;
		sMaintAttrTxt : STRING[13];
		diMaintAttr1 : DINT;
		diMaintAttr2 : DINT;
		wMaintAckLevel : UINT;
		xAckMaint : BOOL;
		xAckFault : BOOL;
		xAckAva : BOOL;
		xAckRead : BOOL;
	END_STRUCT;
END_TYPE
```

#### KGlibMsg.var - Exported constants
```iecst
(********************************************************************
 * COPYRIGHT -- Herbert Kannegiesser GmbH
 ********************************************************************
 * Library: KGlibMsg
 * File: KGlibMsg.var
 * Author: hunholz
 * Created: May 30, 2011
 * Changed: June 15, 2011
 ********************************************************************
 * Constants of library KGlibMsg
 ********************************************************************)
VAR CONSTANT
	MNMSG_CLASS_NO_ACK : USINT := 255;
	MNMSG_CLASS_MAINTENANCE : USINT := 20;
	MNMSG_CLASS_INFO : USINT := 11;
	MNMSG_CLASS_WARNING : USINT := 10;
	MNMSG_CLASS_EXTFAULT : USINT := 1;
	MNMSG_CLASS_INTFAULT : USINT := 0;
	MNMSG_EVENT_COME : UINT := 1;
	MNMSG_EVENT_ACK : UINT := 2;
	MNMSG_EVENT_GONE : UINT := 3;
	MNMSG_EVENT_GONE_TWO : UINT := 4;
	MNMSG_STAT_NOTFOUND : UINT := 1;
	MNMSG_STAT_WRITEPTR : UINT := 2;
	MNMSG_STAT_READPTR : UINT := 3;
	MNMSG_STAT_RBNOREAD : UINT := 10;
	MNMSG_MAX_MSGLIST : UINT := 39;
END_VAR
```

#### KGlibMsg.fun - Exported functions and function blocks
```iecst
(********************************************************************
 * COPYRIGHT -- Herbert Kannegiesser GmbH
 ********************************************************************
 * Library: KGlibMsg
 * File: KGlibMsg.fun
 * Author: hunholz
 * Created: May 30, 2011
 * Changed: June 15, 2011
 ********************************************************************
 * Functions and function blocks of library KGlibMsg
 ********************************************************************)

FUNCTION_BLOCK msgBinSearchCfgList (*Index der Meldung in der Meldungskonfiguration suchen*)
	VAR_INPUT
		MsgCfgList : REFERENCE TO ARRAY[1..65535] OF MsgCfgLine_Typ;
		wCntMsgCfg : UINT;
		wFunctionID : UINT;
		wMsgNo : UINT;
		wInstance : UINT;
	END_VAR
	VAR_OUTPUT
		wMsgIdx : UINT;
		wStatus : UINT;
	END_VAR
	VAR
		dMin : DINT;
		dMax : DINT;
		dSearch : DINT;
	END_VAR
END_FUNCTION_BLOCK

FUNCTION_BLOCK msgInsertMsgLine (*Ein- oder Ausfügen von Meldungen*)
	VAR_INPUT
		AdrIntFaultList : UDINT;
		AdrExtFaultList : UDINT;
		AdrWarnList : UDINT;
		AdrInfoList : UDINT;
		AdrMaintList : UDINT;
		AdrCntIntFault : UDINT;
		AdrCntExtFault : UDINT;
		AdrCntWarn : UDINT;
		AdrCntInfo : UDINT;
		AdrCntMaint : UDINT;
		MsgLine : MsgList_Typ;
		Insert : BOOL;
		Class : USINT;
	END_VAR
	VAR_OUTPUT
		Changed : BOOL;
	END_VAR
	VAR
		MsgList : REFERENCE TO ARRAY[0..MNMSG_MAX_MSGLIST] OF MsgList_Typ;
		bCntList : REFERENCE TO USINT;
		xFound : BOOL;
		i : UINT;
		j : UINT;
		TestCnt : UDINT;
	END_VAR
END_FUNCTION_BLOCK

FUNCTION_BLOCK msgBinSearchTxtLine (*TODO: Add your comment here*)
	VAR_INPUT
		MsgTxtList : REFERENCE TO ARRAY[1..65535] OF MsgTxtLine_Typ;
		wCntMsgTxt : UINT;
		wFunctionID : UINT;
		wNumber : UINT;
		wInstance : UINT := 0;
		bTupel : USINT := 3;
	END_VAR
	VAR_OUTPUT
		wMsgPos : UINT;
		wStatus : UINT;
	END_VAR
	VAR
		xRepeat : BOOL := FALSE;
		xPosFound : BOOL := FALSE;
		xPosFoundLeft : BOOL := FALSE;
		xPosFoundRight : BOOL := FALSE;
		wPos : UINT;
		wPosMin : UINT;
		wPosMax : UINT;
		wPosBeg : UINT;
		wPosEnd : UINT;
		wPosMinLeft : UINT;
		wPosMaxLeft : UINT;
		wPosBegLeft : UINT;
		wPosMinRight : UINT;
		wPosMaxRight : UINT;
		wPosEndRight : UINT;
		wCnt : UINT;
	END_VAR
END_FUNCTION_BLOCK

FUNCTION_BLOCK msgBinSearchHelpTxtLine (*TODO: Add your comment here*)
	VAR_INPUT
		MsgHelpTxtList : REFERENCE TO ARRAY[1..65535] OF MsgHelpTxtLine_Typ;
		wCntMsgHelpTxt : UINT;
		wFunctionID : UINT;
		wNumber : UINT;
		wInstance : UINT := 0;
		bTupel : USINT := 3;
	END_VAR
	VAR_OUTPUT
		wMsgPos : UINT;
		wStatus : UINT;
	END_VAR
	VAR
		xRepeat : BOOL := FALSE;
		xPosFound : BOOL := FALSE;
		xPosFoundLeft : BOOL := FALSE;
		xPosFoundRight : BOOL := FALSE;
		wPos : UINT;
		wPosMin : UINT;
		wPosMax : UINT;
		wPosBeg : UINT;
		wPosEnd : UINT;
		wPosMinLeft : UINT;
		wPosMaxLeft : UINT;
		wPosBegLeft : UINT;
		wPosMinRight : UINT;
		wPosMaxRight : UINT;
		wPosEndRight : UINT;
		wCnt : UINT;
	END_VAR
END_FUNCTION_BLOCK

FUNCTION_BLOCK msgReplSubStr (*TODO: Add your comment here*)
	VAR_INPUT
		utfStr : REFERENCE TO WSTRING[255];
		utfSubStr : REFERENCE TO WSTRING[255];
		utfStrToReplWith : REFERENCE TO WSTRING[255];
		utfStrResult : REFERENCE TO WSTRING[255];
	END_VAR
	VAR_OUTPUT
		wStatus : UINT;
		wMatched : UINT;
	END_VAR
	VAR
		utfStrFirst : WSTRING[1];
		utfStrSecond : WSTRING[1];
		lChrPosStr : UDINT;
		lChrPosSubStr : UDINT;
		xCat : BOOL;
	END_VAR
END_FUNCTION_BLOCK

FUNCTION_BLOCK msgNextChrPos (*TODO: Add your comment here*)
	VAR_INPUT
		utfStr : REFERENCE TO WSTRING[255];
		utfChr : WSTRING[1];
		lStartPos : UDINT;
	END_VAR
	VAR_OUTPUT
		lChrPos : UDINT;
		wStatus : UINT;
	END_VAR
	VAR
		_utfChr : WSTRING[1];
		_lChrPos : UDINT;
		_lUtfLen : UDINT;
	END_VAR
END_FUNCTION_BLOCK
```

#### msgBinSearchCfgList.st - Index der Meldung in der Meldungskonfiguration suchen
```iecst
(********************************************************************
 * COPYRIGHT -- Herbert Kannegiesser GmbH
 ********************************************************************
 * Library: KGlibMsg
 * File: msgBinSearchCfgList.st
 * Author: hunholz
 * Created: May 30, 2011
 * Changed: June 15, 2011
 ********************************************************************
 * Implementation of library KGlibMsg
 ********************************************************************)

(* Index der Meldung in der Meldungskonfiguration suchen *)
FUNCTION_BLOCK msgBinSearchCfgList

	wStatus := MNMSG_STAT_NOTFOUND;
	wMsgIdx := 65535;

	IF wFunctionID = 0 OR wMsgNo = 0 THEN
		RETURN;
	END_IF

	dMin := 1;
	dMax := UINT_TO_DINT(wCntMsgCfg);

	WHILE TRUE DO

		IF dMax < dMin THEN
			// Kein Ergebnis
			wStatus := MNMSG_STAT_NOTFOUND;
			EXIT;
		END_IF

		dSearch := dMin + ((dMax - dMin) / 2);

		IF wFunctionID = MsgCfgList[dSearch].wFunction_ID
			AND wMsgNo = MsgCfgList[dSearch].wMsgNumber
			AND wInstance = MsgCfgList[dSearch].wInstance THEN

			wMsgIdx := DINT_TO_UINT(dSearch);
			wStatus := ERR_OK;

			EXIT;
		END_IF

		IF (wFunctionID > MsgCfgList[dSearch].wFunction_ID) OR
			(wFunctionID = MsgCfgList[dSearch].wFunction_ID
			AND wMsgNo > MsgCfgList[dSearch].wMsgNumber) OR
			(wFunctionID = MsgCfgList[dSearch].wFunction_ID
			AND wMsgNo = MsgCfgList[dSearch].wMsgNumber
			AND wInstance > MsgCfgList[dSearch].wInstance) THEN

				dMin := dSearch + 1;

		ELSE

				dMax := dSearch - 1;

		END_IF

	END_WHILE;

END_FUNCTION_BLOCK
```

#### msgInsertMsgLine.st - Ein- oder Ausfügen von Meldungen
```iecst
(********************************************************************
 * COPYRIGHT -- Herbert Kannegiesser GmbH
 ********************************************************************
 * Library: KGlibMsg
 * File: msgInsertMsgLine.st
 * Author: hunholz
 * Created: May 30, 2011
 * Changed: June 15, 2011
 ********************************************************************
 * Implementation of library KGlibMsg
 ********************************************************************)

(* Ein- oder Ausfügen von Meldungen *)
FUNCTION_BLOCK msgInsertMsgLine

	TestCnt := TestCnt + 1;

	Changed := FALSE;

	// VAR Ref MsgList of MsgList_Typ[0..MSGLISTMAX]
	// Constant UINT MSGLISTMAX = 39
	// VAR_INPUT USINT Class belongs to KGlibMsg
	// Constant USINT MSG_CLASS_INTFAULT = 0
	// VAR_INPUT UDINT AdrIntFaultList, AdrCntIntFault
	IF Class = MNMSG_CLASS_INTFAULT AND AdrIntFaultList <> 0 AND AdrCntIntFault <> 0 THEN
		MsgList ACCESS AdrIntFaultList;
		bCntList ACCESS AdrCntIntFault;
	ELSIF Class = MNMSG_CLASS_EXTFAULT AND AdrExtFaultList <> 0 AND AdrCntExtFault <> 0 THEN
		MsgList ACCESS AdrExtFaultList;
		bCntList ACCESS AdrCntExtFault;
	ELSIF Class = MNMSG_CLASS_WARNING AND AdrWarnList <> 0 AND AdrCntWarn <> 0 THEN
		MsgList ACCESS AdrWarnList;
		bCntList ACCESS AdrCntWarn;
	ELSIF Class = MNMSG_CLASS_INFO AND AdrInfoList <> 0 AND AdrCntInfo <> 0 THEN
		MsgList ACCESS AdrInfoList;
		bCntList ACCESS  AdrCntInfo;
	ELSIF Class = MNMSG_CLASS_MAINTENANCE AND AdrMaintList <> 0 THEN
		MsgList ACCESS AdrMaintList;
		bCntList ACCESS AdrCntMaint;
	ELSE
		RETURN;
	END_IF

	xFound := FALSE;

	// VAR Ref USINT bCntList
	// VAR Ref MsgList of MsgList_Typ[0..MSGLISTMAX]
	// Constant UINT MSGLISTMAX = 39

	IF bCntList > 0 THEN

		FOR i := 0 TO bCntList-1	DO
			IF MsgList[i].wFunction_ID = MsgLine.wFunction_ID AND MsgList[i].wMsgNumber = MsgLine.wMsgNumber AND MsgList[i].bInstance = MsgLine.bInstance THEN

				// DINT brsmemcmp 'compares memory areas' belongs to library AsBrStr
				// VAR_INPUT MsgLine of MsgList_Typ
				IF Insert  AND brsmemcmp(ADR(MsgList[i]),ADR(MsgLine),SIZEOF(MsgLine)) <> 0 THEN
					MsgList[i] := MsgLine;
					Changed := TRUE;
				END_IF

				xFound := TRUE;
				EXIT;

			END_IF

		END_FOR

	END_IF

	IF Insert THEN	// xInsert ?
		// Hinzufügen

		IF NOT xFound AND bCntList <= MNMSG_MAX_MSGLIST THEN
			MsgList[bCntList] := MsgLine;
			bCntList := bCntList + 1;
			Changed := TRUE;
		END_IF

	ELSE
		// Eintrag entfernen
		// UDINT brsmemset 'fills the memory area with specific values'
		// VAR Ref USINT bCntList
		IF xFound THEN

			brsmemset(ADR(MsgList[MNMSG_MAX_MSGLIST]),0,SIZEOF(MsgList[MNMSG_MAX_MSGLIST]));

			FOR j := i TO bCntList-1 DO
				IF j <> MNMSG_MAX_MSGLIST THEN
					MsgList[j] := MsgList[j+1];
				END_IF
			END_FOR

			bCntList := bCntList - 1;

			Changed := TRUE;

		END_IF

	END_IF

END_FUNCTION_BLOCK
```

#### msgBinSearchTxtLine.st
```iecst
(********************************************************************
 * COPYRIGHT -- Herbert Kannegiesser GmbH
 ********************************************************************
 * Library: KGlibMsg
 * File: msgBinSearchTxtLine.st
 * Author: kuehne
 * Created: November 29, 2011
 ********************************************************************
 * Implementation of library KGlibMsg
 ********************************************************************)

(* TODO: Add your comment here *)
FUNCTION_BLOCK msgBinSearchTxtLine
	wStatus := MNMSG_STAT_NOTFOUND;
	wMsgPos := 65535;
	IF bTupel = 0 OR bTupel > 3 THEN
		RETURN;
	END_IF;
	IF bTupel = 1 THEN
		IF (wFunctionID < 1) OR (wCntMsgTxt < 1) THEN
			RETURN;
		END_IF;
	END_IF;
	IF bTupel = 2 OR bTupel = 3 THEN
		IF (wFunctionID < 1) OR (wNumber < 1) OR (wCntMsgTxt < 1) THEN
			RETURN;
		END_IF;
	END_IF;
	wPosMin := 0;
	wPosBeg := wPosMin;
	wPosEnd := wPosMin + wCntMsgTxt - 1;
	IF wPosEnd = wPosBeg THEN
		CASE bTupel OF
			1:
				IF (MsgTxtList[wPosBeg].wFunctionID = wFunctionID) THEN
					wMsgPos := wPosBeg;
					wStatus := ERR_OK;
					RETURN;
				ELSE
					RETURN;
				END_IF;
			2:
				IF (MsgTxtList[wPosBeg].wFunctionID = wFunctionID) AND (MsgTxtList[wPosBeg].wNumber = wNumber) THEN
					wMsgPos := wPosBeg;
					wStatus := ERR_OK;
					RETURN;
				ELSE
					RETURN;
				END_IF;
			3:
				IF (MsgTxtList[wPosBeg].wFunctionID = wFunctionID) AND (MsgTxtList[wPosBeg].wNumber = wNumber) AND ((MsgTxtList[wPosBeg].wInstance = wInstance) OR (wInstance = 0)) THEN
					wMsgPos := wPosBeg;
					wStatus := ERR_OK;
					RETURN;
				ELSE
					RETURN;
				END_IF;
		END_CASE;
	END_IF;
	wPosMin := 1;
	wPosBeg := wPosMin;
	wPosMax := wPosMin + wCntMsgTxt - 1;
	wPosEnd := wPosMin + wCntMsgTxt - 1;
	wPos := (wPosMin + wPosMax) / 2;
	xPosFound := FALSE;
	WHILE NOT xPosFound DO
		IF ((wPos = (wPosBeg + 1)) OR (wPos = wPosBeg)) AND NOT xPosFound THEN
			wPos := wPosBeg;
			IF (MsgTxtList[wPos].wFunctionID > wFunctionID) AND (MsgTxtList[wPos + 1].wFunctionID > wFunctionID) THEN
				wPos := wPosBeg + 0;
				xPosFound := TRUE;
			ELSIF (MsgTxtList[wPos].wFunctionID < wFunctionID) AND (MsgTxtList[wPos + 1].wFunctionID > wFunctionID) THEN
				wPos := wPosBeg + 1;
				xPosFound := TRUE;
			ELSIF (MsgTxtList[wPos].wFunctionID < wFunctionID) AND (MsgTxtList[wPos + 1].wFunctionID = wFunctionID) THEN
				wPos := wPosBeg + 1;
				xPosFound := TRUE;
			ELSIF (MsgTxtList[wPos].wFunctionID < wFunctionID) AND (MsgTxtList[wPos + 1].wFunctionID < wFunctionID) THEN
				IF wPosEnd = (wPosBeg + 1) THEN
					wCnt := wPosBeg;
					WHILE MsgTxtList[wCnt].wFunctionID < wFunctionID AND (wCnt < wPosEnd) DO
						wCnt := wCnt + 1;
					END_WHILE;
					wPos := wCnt;
				ELSE
					wPos := wPosBeg + 2;
					IF NOT (MsgTxtList[wPos].wFunctionID = wFunctionID) THEN
						wCnt := wPosBeg;
						WHILE MsgTxtList[wCnt].wFunctionID < wFunctionID AND (wCnt < wPosEnd) DO
							wCnt := wCnt + 1;
						END_WHILE;
						wPos := wCnt;
					END_IF;
				END_IF;
				xPosFound := TRUE;
			ELSIF (MsgTxtList[wPos].wFunctionID = wFunctionID) AND (MsgTxtList[wPos + 1].wFunctionID > wFunctionID) THEN
				wPos := wPosBeg + 0;
				xPosFound := TRUE;
			ELSIF (MsgTxtList[wPos].wFunctionID = wFunctionID) AND (MsgTxtList[wPos + 1].wFunctionID = wFunctionID) THEN
				wPos := wPosBeg + 0;
				xPosFound := TRUE;
			ELSE
				// to be sure: implement a simple algorithm with linear time here to avoid unlimited repetition
				wCnt := wPosBeg;
				WHILE MsgTxtList[wCnt].wFunctionID < wFunctionID AND (wCnt < wPosEnd) DO
					wCnt := wCnt + 1;
				END_WHILE;
				wPos := wCnt;
				xPosFound := TRUE;
			END_IF;
		END_IF;
		IF ((wPos = (wPosEnd - 1)) OR (wPos = wPosEnd)) AND NOT xPosFound THEN
			wPos := wPosEnd;
			IF (MsgTxtList[wPos].wFunctionID < wFunctionID) AND (MsgTxtList[wPos - 1].wFunctionID < wFunctionID) THEN
				wPos := wPosEnd;
				xPosFound := TRUE;
			ELSIF (MsgTxtList[wPos].wFunctionID > wFunctionID) AND (MsgTxtList[wPos - 1].wFunctionID < wFunctionID) THEN
				wPos := wPosEnd - 0;
				xPosFound := TRUE;
			ELSIF (MsgTxtList[wPos].wFunctionID > wFunctionID) AND (MsgTxtList[wPos - 1].wFunctionID = wFunctionID) THEN
				wPos := wPosEnd - 1;
				xPosFound := TRUE;
			(* ELSIF (MsgTxtList[wPos].wFunctionID > wFunctionID) AND (MsgTxtList[wPos - 1].wFunctionID > wFunctionID) THEN
				wPos := wPosEnd - 1;
				xPosFound := TRUE; *)
			ELSIF (MsgTxtList[wPos].wFunctionID = wFunctionID) AND (MsgTxtList[wPos - 1].wFunctionID < wFunctionID) THEN
				wPos := wPosEnd - 0;
				xPosFound := TRUE;
			ELSIF (MsgTxtList[wPos].wFunctionID = wFunctionID) AND (MsgTxtList[wPos - 1].wFunctionID = wFunctionID) THEN
				wPos := wPosEnd - 1;
				xPosFound := TRUE;
			ELSE
				// to be sure: implement a simple algorithm with linear time here to avoid unlimited repetition
				wCnt := wPosBeg;
				WHILE MsgTxtList[wCnt].wFunctionID < wFunctionID AND (wCnt < wPosEnd) DO
					wCnt := wCnt + 1;
				END_WHILE;
				wPos := wCnt;
				xPosFound := TRUE;
			END_IF;
		END_IF;
		IF NOT xPosFound THEN
			IF (MsgTxtList[wPos].wFunctionID > wFunctionID) AND (MsgTxtList[wPos + 1].wFunctionID > wFunctionID) THEN
				wPosMax := wPos;
				wPos := (wPosMin + wPosMax) / 2;
				IF (wPosMax - wPos) = 0 THEN
					wCnt := wPosBeg;
					WHILE MsgTxtList[wCnt].wFunctionID < wFunctionID AND (wCnt < wPosEnd) DO
						wCnt := wCnt + 1;
					END_WHILE;
					wPos := wCnt;
					xPosFound := TRUE;
				END_IF;
			ELSIF (MsgTxtList[wPos].wFunctionID < wFunctionID) AND (MsgTxtList[wPos + 1].wFunctionID < wFunctionID) THEN
				wPosMin := wPos;
				wPos := (wPosMin + wPosMax) / 2;
				IF (wPos - wPosMin) = 0 THEN
					wCnt := wPosBeg;
					WHILE MsgTxtList[wCnt].wFunctionID < wFunctionID AND (wCnt < wPosEnd) DO
						wCnt := wCnt + 1;
					END_WHILE;
					wPos := wCnt;
					xPosFound := TRUE;
				END_IF;
			ELSIF (MsgTxtList[wPos].wFunctionID < wFunctionID) AND (MsgTxtList[wPos + 1].wFunctionID > wFunctionID) THEN
				xPosFound := TRUE;
				wPos := wPos + 1;
			ELSIF (MsgTxtList[wPos].wFunctionID < wFunctionID) AND (MsgTxtList[wPos + 1].wFunctionID = wFunctionID) THEN
				xPosFound := TRUE;
				wPos := wPos + 1;
			ELSIF (MsgTxtList[wPos].wFunctionID = wFunctionID) AND (MsgTxtList[wPos + 1].wFunctionID > wFunctionID) THEN
				xPosFound := TRUE;
				wPos := wPos;
			ELSIF (MsgTxtList[wPos].wFunctionID = wFunctionID) AND (MsgTxtList[wPos + 1].wFunctionID = wFunctionID) THEN
				xPosFound := TRUE;
				wPos := wPos;
			ELSE
				// to be sure: implement a simple algorithm with linear time here to avoid unlimited repetition
				wCnt := wPosBeg;
				WHILE MsgTxtList[wCnt].wFunctionID < wFunctionID AND (wCnt < wPosEnd) DO
					wCnt := wCnt + 1;
				END_WHILE;
				wPos := wCnt;
				xPosFound := TRUE;
			END_IF;
		END_IF;
	END_WHILE;
	IF MsgTxtList[wPos].wFunctionID <> wFunctionID THEN
		wPosMin := wPosBeg;
		wPosMax := wPosEnd;
		wCnt := wPosBeg;
		WHILE MsgTxtList[wCnt].wFunctionID <> wFunctionID AND (wCnt < wPosEnd) DO
			wCnt := wCnt + 1;
		END_WHILE;
		wPos := wCnt;
		xPosFound := TRUE;
	END_IF;
	IF bTupel = 1 THEN
		IF MsgTxtList[wPos].wFunctionID = wFunctionID THEN
			wMsgPos := wPos;
			wStatus := ERR_OK;
			RETURN;
		ELSE
			RETURN;
		END_IF;
	END_IF;
	IF MsgTxtList[wPos].wFunctionID = wFunctionID THEN
		//###DK2011Dec07
		wPosMinLeft := wPosMin;
		wPosMaxLeft := wPos;
		wPosBegLeft := (wPosMinLeft + wPosMaxLeft) / 2;
		xPosFoundLeft := FALSE;
		xRepeat := TRUE;
		WHILE (NOT xPosFoundLeft) AND xRepeat DO
			IF ((wPosBegLeft = (wPosBeg + 1)) OR (wPosBegLeft = wPosBeg)) AND (NOT xPosFoundLeft) AND xRepeat THEN
				wPosBegLeft := wPosBeg;
				IF (MsgTxtList[wPosBegLeft].wFunctionID = wFunctionID) AND (MsgTxtList[wPosBegLeft + 1].wFunctionID = wFunctionID) THEN
					xPosFoundLeft := TRUE;
					xRepeat := FALSE;
				ELSIF (MsgTxtList[wPosBegLeft].wFunctionID < wFunctionID) AND (MsgTxtList[wPosBegLeft + 1].wFunctionID = wFunctionID) THEN
					wPosBegLeft := wPosBeg + 1;
					xPosFoundLeft := TRUE;
					xRepeat := FALSE;
				ELSE
					xPosFoundLeft := FALSE;
					xRepeat := FALSE;
				END_IF;
			END_IF;
			IF (NOT xPosFoundLeft) AND xRepeat THEN
				IF (MsgTxtList[wPosBegLeft].wFunctionID = wFunctionID) AND (MsgTxtList[wPosBegLeft - 1].wFunctionID = wFunctionID) THEN
					wPosMaxLeft := wPosBegLeft;
					wPosBegLeft := (wPosMinLeft + wPosMaxLeft) / 2;
					IF (wPosMaxLeft - wPosBegLeft) = 0 THEN
						xPosFoundLeft := FALSE;
						xRepeat := FALSE;
					END_IF;
				ELSIF (MsgTxtList[wPosBegLeft].wFunctionID < wFunctionID) AND (MsgTxtList[wPosBegLeft - 1].wFunctionID < wFunctionID) THEN
					wPosMinLeft := wPosBegLeft;
					wPosBegLeft := (wPosMinLeft + wPosMaxLeft) / 2;
					IF (wPosMinLeft - wPosBegLeft) = 0 THEN
						xPosFoundLeft := FALSE;
						xRepeat := FALSE;
					END_IF;
				ELSIF (MsgTxtList[wPosBegLeft].wFunctionID = wFunctionID) AND (MsgTxtList[wPosBegLeft - 1].wFunctionID < wFunctionID) THEN
					xPosFoundLeft := TRUE;
					xRepeat := FALSE;
				ELSE
					xPosFoundLeft := FALSE;
					xRepeat := FALSE;
				END_IF;
			END_IF;
		END_WHILE;
		//###DK2011Dec07
		//###DK2011Dec07
		wPosMinRight := wPos;
		wPosMaxRight := wPosMax;
		wPosEndRight := (wPosMinRight + wPosMaxRight) / 2;
		xPosFoundRight := FALSE;
		xRepeat := TRUE;
		WHILE (NOT xPosFoundRight) AND xRepeat DO
			IF ((wPosEndRight = (wPosEnd - 1)) OR (wPosEndRight = wPosEnd)) AND (NOT xPosFoundRight) AND xRepeat THEN
				wPosEndRight := wPosEnd;
				IF (MsgTxtList[wPosEndRight].wFunctionID = wFunctionID) AND (MsgTxtList[wPosEndRight - 1].wFunctionID = wFunctionID) THEN
					xPosFoundRight := TRUE;
					xRepeat := FALSE;
				ELSIF (MsgTxtList[wPosEndRight].wFunctionID > wFunctionID) AND (MsgTxtList[wPosEndRight - 1].wFunctionID = wFunctionID) THEN
					wPosEndRight := wPosEnd - 1;
					xPosFoundRight := TRUE;
					xRepeat := FALSE;
				ELSE
					xPosFoundRight := FALSE;
					xRepeat := FALSE;
				END_IF;
			END_IF;
			IF (NOT xPosFoundRight) AND xRepeat THEN
				IF (MsgTxtList[wPosEndRight].wFunctionID = wFunctionID) AND (MsgTxtList[wPosEndRight + 1].wFunctionID = wFunctionID) THEN
					wPosMinRight := wPosEndRight;
					wPosEndRight := (wPosMinRight + wPosMaxRight) / 2;
					IF (wPosMinRight - wPosEndRight) = 0 THEN
						xPosFoundRight := FALSE;
						xRepeat := FALSE;
					END_IF;
				ELSIF (MsgTxtList[wPosEndRight].wFunctionID > wFunctionID) AND (MsgTxtList[wPosEndRight + 1].wFunctionID > wFunctionID) THEN
					wPosMaxRight := wPosEndRight;
					wPosEndRight := (wPosMinRight + wPosMaxRight) / 2;
					IF (wPosMaxRight - wPosEndRight) = 0 THEN
						xPosFoundRight := FALSE;
						xRepeat := FALSE;
					END_IF;
				ELSIF (MsgTxtList[wPosEndRight].wFunctionID = wFunctionID) AND (MsgTxtList[wPosEndRight + 1].wFunctionID > wFunctionID) THEN
					xPosFoundRight := TRUE;
					xRepeat := FALSE;
				ELSE
					xPosFoundRight := FALSE;
					xRepeat := FALSE;
				END_IF;
			END_IF;
		END_WHILE;
		//###DK2011Dec07
		IF NOT xPosFoundLeft THEN
			wPosBeg := wPos;
			IF (wPosBeg - 1) >= wPosMin THEN
				IF MsgTxtList[wPosBeg - 1].wFunctionID = wFunctionID THEN
					wPosBeg := wPosBeg - 1;
					xRepeat := TRUE;
				ELSE
					xRepeat := FALSE;
				END_IF;
			ELSE
				xRepeat := FALSE;
			END_IF;
			WHILE xRepeat DO
				IF (wPosBeg - 1) >= wPosMin THEN
					IF MsgTxtList[wPosBeg - 1].wFunctionID = wFunctionID THEN
						wPosBeg := wPosBeg - 1;
						xRepeat := TRUE;
					ELSE
						xRepeat := FALSE;
					END_IF;
				ELSE
					xRepeat := FALSE;
				END_IF;
			END_WHILE;
		ELSE
			wPosBeg := wPosBegLeft;
		END_IF;
		IF NOT xPosFoundRight THEN
			wPosEnd := wPos;
			IF (wPosEnd + 1) <= (wPosMin + wCntMsgTxt - 1) THEN
				IF MsgTxtList[wPosEnd + 1].wFunctionID = wFunctionID THEN
					wPosEnd := wPosEnd + 1;
					xRepeat := TRUE;
				ELSE
					xRepeat := FALSE;
				END_IF;
			ELSE
				xRepeat := FALSE;
			END_IF;
			WHILE xRepeat DO
				IF (wPosEnd + 1) <= (wPosMin + wCntMsgTxt - 1) THEN
					IF MsgTxtList[wPosEnd + 1].wFunctionID = wFunctionID THEN
						wPosEnd := wPosEnd + 1;
						xRepeat := TRUE;
					ELSE
						xRepeat := FALSE;
					END_IF;
				ELSE
					xRepeat := FALSE;
				END_IF;
			END_WHILE;
		ELSE
			wPosEnd := wPosEndRight;
		END_IF;
	ELSE
		RETURN;
	END_IF;
	wPosMin := wPosBeg;
	wPosMax := wPosEnd;
	wPos := (wPosMin + wPosMax) / 2;
	xPosFound := FALSE;
	IF wPosMax = wPosBeg THEN
		wPos := wPosBeg;
		xPosFound := TRUE;
	END_IF;
	WHILE NOT xPosFound DO
		IF ((wPos = (wPosBeg + 1)) OR (wPos = wPosBeg)) AND NOT xPosFound THEN
			wPos := wPosBeg;
			IF (MsgTxtList[wPos].wNumber > wNumber) AND (MsgTxtList[wPos + 1].wNumber > wNumber) THEN
				wPos := wPosBeg + 0;
				xPosFound := TRUE;
			ELSIF (MsgTxtList[wPos].wNumber < wNumber) AND (MsgTxtList[wPos + 1].wNumber > wNumber) THEN
				wPos := wPosBeg + 1;
				xPosFound := TRUE;
			ELSIF (MsgTxtList[wPos].wNumber < wNumber) AND (MsgTxtList[wPos + 1].wNumber = wNumber) THEN
				wPos := wPosBeg + 1;
				xPosFound := TRUE;
			ELSIF (MsgTxtList[wPos].wNumber < wNumber) AND (MsgTxtList[wPos + 1].wNumber < wNumber) THEN
				IF wPosEnd = (wPosBeg + 1) THEN
					wCnt := wPosBeg;
					WHILE MsgTxtList[wCnt].wNumber < wNumber AND (wCnt < wPosEnd) DO
						wCnt := wCnt + 1;
					END_WHILE;
					wPos := wCnt;
				ELSE
					wPos := wPosBeg + 2;
					IF NOT (MsgTxtList[wPos].wNumber = wNumber) THEN
						wCnt := wPosBeg;
						WHILE MsgTxtList[wCnt].wNumber < wNumber AND (wCnt < wPosEnd) DO
							wCnt := wCnt + 1;
						END_WHILE;
						wPos := wCnt;
					END_IF;
				END_IF;
				xPosFound := TRUE;
			ELSIF (MsgTxtList[wPos].wNumber = wNumber) AND (MsgTxtList[wPos + 1].wNumber > wNumber) THEN
				wPos := wPosBeg + 0;
				xPosFound := TRUE;
			ELSIF (MsgTxtList[wPos].wNumber = wNumber) AND (MsgTxtList[wPos + 1].wNumber = wNumber) THEN
				wPos := wPosBeg + 0;
				xPosFound := TRUE;
			ELSE
				// to be sure: implement a simple algorithm with linear time here to avoid unlimited repetition
				wCnt := wPosBeg;
				WHILE MsgTxtList[wCnt].wNumber < wNumber AND (wCnt < wPosEnd) DO
					wCnt := wCnt + 1;
				END_WHILE;
				wPos := wCnt;
				xPosFound := TRUE;
			END_IF;
		END_IF;
		IF ((wPos = (wPosEnd - 1)) OR (wPos = wPosEnd)) AND NOT xPosFound THEN
			wPos := wPosEnd;
			IF (MsgTxtList[wPos].wNumber < wNumber) AND (MsgTxtList[wPos - 1].wNumber < wNumber) THEN
				wPos := wPosEnd;
				xPosFound := TRUE;
			ELSIF (MsgTxtList[wPos].wNumber > wNumber) AND (MsgTxtList[wPos - 1].wNumber < wNumber) THEN
				wPos := wPosEnd - 0;
				xPosFound := TRUE;
			ELSIF (MsgTxtList[wPos].wNumber > wNumber) AND (MsgTxtList[wPos - 1].wNumber = wNumber) THEN
				wPos := wPosEnd - 1;
				xPosFound := TRUE;
			(* ELSIF (MsgTxtList[wPos].wNumber > wNumber) AND (MsgTxtList[wPos - 1].wNumber > wNumber) THEN
				wPos := wPosEnd - 1;
				xPosFound := TRUE; *)
			ELSIF (MsgTxtList[wPos].wNumber = wNumber) AND (MsgTxtList[wPos - 1].wNumber < wNumber) THEN
				wPos := wPosEnd - 0;
				xPosFound := TRUE;
			ELSIF (MsgTxtList[wPos].wNumber = wNumber) AND (MsgTxtList[wPos - 1].wNumber = wNumber) THEN
				wPos := wPosEnd - 1;
				xPosFound := TRUE;
			ELSE
				// to be sure: implement a simple algorithm with linear time here to avoid unlimited repetition
				wCnt := wPosBeg;
				WHILE MsgTxtList[wCnt].wNumber < wNumber AND (wCnt < wPosEnd) DO
					wCnt := wCnt + 1;
				END_WHILE;
				wPos := wCnt;
				xPosFound := TRUE;
			END_IF;
		END_IF;
		IF NOT xPosFound THEN
			IF (MsgTxtList[wPos].wNumber > wNumber) AND (MsgTxtList[wPos + 1].wNumber > wNumber) THEN
				wPosMax := wPos;
				wPos := (wPosMin + wPosMax) / 2;
				IF (wPosMax - wPos) = 0 THEN
					wCnt := wPosBeg;
					WHILE MsgTxtList[wCnt].wNumber < wNumber AND (wCnt < wPosEnd) DO
						wCnt := wCnt + 1;
					END_WHILE;
					wPos := wCnt;
					xPosFound := TRUE;
				END_IF;
			ELSIF (MsgTxtList[wPos].wNumber < wNumber) AND (MsgTxtList[wPos + 1].wNumber < wNumber) THEN
				wPosMin := wPos;
				wPos := (wPosMin + wPosMax) / 2;
				IF (wPos - wPosMin) = 0 THEN
					wCnt := wPosBeg;
					WHILE MsgTxtList[wCnt].wNumber < wNumber AND (wCnt < wPosEnd) DO
						wCnt := wCnt + 1;
					END_WHILE;
					wPos := wCnt;
					xPosFound := TRUE;
				END_IF;
			ELSIF (MsgTxtList[wPos].wNumber < wNumber) AND (MsgTxtList[wPos + 1].wNumber > wNumber) THEN
				xPosFound := TRUE;
				wPos := wPos + 1;
			ELSIF (MsgTxtList[wPos].wNumber < wNumber) AND (MsgTxtList[wPos + 1].wNumber = wNumber) THEN
				xPosFound := TRUE;
				wPos := wPos + 1;
			ELSIF (MsgTxtList[wPos].wNumber = wNumber) AND (MsgTxtList[wPos + 1].wNumber > wNumber) THEN
				xPosFound := TRUE;
				wPos := wPos;
			ELSIF (MsgTxtList[wPos].wNumber = wNumber) AND (MsgTxtList[wPos + 1].wNumber = wNumber) THEN
				xPosFound := TRUE;
				wPos := wPos;
			ELSE
				// to be sure: implement a simple algorithm with linear time here to avoid unlimited repetition
				wCnt := wPosBeg;
				WHILE MsgTxtList[wCnt].wNumber < wNumber AND (wCnt < wPosEnd) DO
					wCnt := wCnt + 1;
				END_WHILE;
				wPos := wCnt;
				xPosFound := TRUE;
			END_IF;
		END_IF;
	END_WHILE;
	IF MsgTxtList[wPos].wNumber <> wNumber THEN
		wPosMin := wPosBeg;
		wPosMax := wPosEnd;
		wCnt := wPosBeg;
		WHILE MsgTxtList[wCnt].wNumber <> wNumber AND (wCnt < wPosEnd) DO
			wCnt := wCnt + 1;
		END_WHILE;
		wPos := wCnt;
		xPosFound := TRUE;
	END_IF;
	IF MsgTxtList[wPos].wNumber <> wNumber THEN
		RETURN;
	END_IF;
	IF wInstance = 0 OR bTupel = 2 THEN
		wMsgPos := wPos;
		wStatus := ERR_OK;
		RETURN;
	END_IF;
	wPosBeg := wPos;
	wPosEnd := wPos;
	IF (wPosBeg - 1) >= wPosMin THEN
		IF MsgTxtList[wPosBeg - 1].wNumber = wNumber THEN
			wPosBeg := wPosBeg - 1;
			xRepeat := TRUE;
		ELSE
			xRepeat := FALSE;
		END_IF;
	ELSE
		xRepeat := FALSE;
	END_IF;
	WHILE xRepeat DO
		IF (wPosBeg - 1) >= wPosMin THEN
			IF MsgTxtList[wPosBeg - 1].wNumber = wNumber THEN
				wPosBeg := wPosBeg - 1;
				xRepeat := TRUE;
			ELSE
				xRepeat := FALSE;
			END_IF;
		ELSE
			xRepeat := FALSE;
		END_IF;
	END_WHILE;
	IF (wPosEnd + 1) <= wPosMax THEN
		IF MsgTxtList[wPosEnd + 1].wNumber = wNumber THEN
			wPosEnd := wPosEnd + 1;
			xRepeat := TRUE;
		ELSE
			xRepeat := FALSE;
		END_IF;
	ELSE
		xRepeat := FALSE;
	END_IF;
	WHILE xRepeat DO
		IF (wPosEnd + 1) <= wPosMax THEN
			IF MsgTxtList[wPosEnd + 1].wNumber = wNumber THEN
				wPosEnd := wPosEnd + 1;
				xRepeat := TRUE;
			ELSE
				xRepeat := FALSE;
			END_IF;
		ELSE
			xRepeat := FALSE;
		END_IF;
	END_WHILE;
	wCnt := wPosBeg;
	WHILE MsgTxtList[wCnt].wInstance <> wInstance AND (wCnt < wPosEnd) DO
		wCnt := wCnt + 1;
	END_WHILE;
	wPos := wCnt;
	IF MsgTxtList[wPos].wInstance = wInstance THEN
		wMsgPos := wPos;
		wStatus := ERR_OK;
	END_IF;
END_FUNCTION_BLOCK
```
